LIN {X 0,Y 411.233,Z 499.748,A -85,B 0,C 180,E1 -10713.92,E2 -10713.92} C_VEL
LIN {X 0,Y 411.528,Z 496.938,A -85,B 0,C 180,E1 -10715.39,E2 -10715.39} C_VEL
LIN {X 0,Y 411.956,Z 493.12,A -85,B 0,C 180,E1 -10716.859,E2 -10716.859} C_VEL
LIN {X 0,Y 412.248,Z 487.246,A -85,B 0,C 180,E1 -10718.588,E2 -10718.588} C_VEL
LIN {X 0,Y 412.886,Z 480.826,A -85,B 0,C 180,E1 -10720.048,E2 -10720.048} C_VEL
LIN {X 0,Y 413.463,Z 474.571,A -85,B 0,C 180,E1 -10721.218,E2 -10721.218} C_VEL
LIN {X 0,Y 413.16,Z 470.905,A -85,B 0,C 180,E1 -10721.852,E2 -10721.852} C_VEL
LIN {X 0,Y 410.83,Z 464.808,A -85,B 0,C 180,E1 -10722.887,E2 -10722.887} C_VEL
LIN {X 0,Y 408.489,Z 458.169,A -85,B 0,C 180,E1 -10723.864,E2 -10723.864} C_VEL
LIN {X 0,Y 408.169,Z 453.615,A -85,B 0,C 180,E1 -10724.401,E2 -10724.401} C_VEL
LIN {X 0,Y 408.88,Z 442.463,A -85,B 0,C 180,E1 -10725.449,E2 -10725.449} C_VEL
LIN {X 0,Y 409.109,Z 437.491,A -85,B 0,C 180,E1 -10725.842,E2 -10725.842} C_VEL
LIN {X 0,Y 406.256,Z 427.518,A -85,B 0,C 180,E1 -10726.674,E2 -10726.674} C_VEL
LIN {X 0,Y 404.21,Z 421.137,A -85,B 0,C 180,E1 -10727.15,E2 -10727.15} C_VEL
LIN {X 0,Y 404.167,Z 421.143,A -85,B 0,C 180,E1 -10730.351,E2 -10730.351} C_VEL
LIN {X 0,Y 404.172,Z 421.141,A -85,B 0,C 180,E1 -10733.574,E2 -10733.574} C_VEL
LIN {X 0,Y 404.187,Z 421.137,A -85,B 0,C 180,E1 -10735.766,E2 -10735.766} C_VEL
LIN {X 0,Y 404.198,Z 421.134,A -85,B 0,C 180,E1 -10737.999,E2 -10737.999} C_VEL
LIN {X 0,Y 404.142,Z 421.144,A -85,B 0,C 180,E1 -10741.558,E2 -10741.558} C_VEL
LIN {X 0,Y 404.188,Z 421.14,A -85,B 0,C 180,E1 -10745.016,E2 -10745.016} C_VEL
LIN {X 0,Y 404.167,Z 421.141,A -85,B 0,C 180,E1 -10748.756,E2 -10748.756} C_VEL
LIN {X 0,Y 404.194,Z 421.136,A -85,B 0,C 180,E1 -10751.611,E2 -10751.611} C_VEL
LIN {X 0,Y 404.194,Z 421.136,A -85,B 0,C 180,E1 -10754.529,E2 -10754.529} C_VEL
LIN {X 0,Y 404.142,Z 421.144,A -85,B 0,C 180,E1 -10757.296,E2 -10757.296} C_VEL
LIN {X 0,Y 404.171,Z 421.138,A -85,B 0,C 180,E1 -10759.955,E2 -10759.955} C_VEL
LIN {X 0,Y 404.139,Z 421.146,A -85,B 0,C 180,E1 -10763.125,E2 -10763.125} C_VEL
LIN {X 0,Y 404.147,Z 421.141,A -85,B 0,C 180,E1 -10766.188,E2 -10766.188} C_VEL
LIN {X 0,Y 404.148,Z 421.14,A -85,B 0,C 180,E1 -10769.715,E2 -10769.715} C_VEL
LIN {X 0,Y 404.197,Z 421.137,A -85,B 0,C 180,E1 -10773.123,E2 -10773.123} C_VEL
LIN {X 0,Y 404.179,Z 421.138,A -85,B 0,C 180,E1 -10775.334,E2 -10775.334} C_VEL
LIN {X 0,Y 404.141,Z 421.146,A -85,B 0,C 180,E1 -10778.581,E2 -10778.581} C_VEL
LIN {X 0,Y 404.213,Z 421.132,A -85,B 0,C 180,E1 -10781.762,E2 -10781.762} C_VEL
LIN {X 0,Y 404.211,Z 421.136,A -85,B 0,C 180,E1 -10784.882,E2 -10784.882} C_VEL
LIN {X 0,Y 404.273,Z 421.126,A -85,B 0,C 180,E1 -10787.959,E2 -10787.959} C_VEL
LIN {X 0,Y 404.27,Z 421.127,A -85,B 0,C 180,E1 -10790.998,E2 -10790.998} C_VEL
LIN {X 0,Y 404.421,Z 421.109,A -85,B 0,C 180,E1 -10794.015,E2 -10794.015} C_VEL
LIN {X 0,Y 404.486,Z 421.101,A -85,B 0,C 180,E1 -10798.008,E2 -10798.008} C_VEL
LIN {X 0,Y 404.615,Z 421.084,A -85,B 0,C 180,E1 -10800,E2 -10800} C_VEL
LIN {X 0,Y 404.427,Z 421.107,A -85,B 0,C 180,E1 -10802.988,E2 -10802.988} C_VEL
LIN {X 0,Y 404.421,Z 421.11,A -85,B 0,C 180,E1 -10805.985,E2 -10805.985} C_VEL
LIN {X 0,Y 404.269,Z 421.126,A -85,B 0,C 180,E1 -10809.001,E2 -10809.001} C_VEL
LIN {X 0,Y 404.272,Z 421.129,A -85,B 0,C 180,E1 -10812.041,E2 -10812.041} C_VEL
LIN {X 0,Y 404.211,Z 421.132,A -85,B 0,C 180,E1 -10815.118,E2 -10815.118} C_VEL
LIN {X 0,Y 404.213,Z 421.137,A -85,B 0,C 180,E1 -10818.238,E2 -10818.238} C_VEL
LIN {X 0,Y 404.141,Z 421.142,A -85,B 0,C 180,E1 -10821.419,E2 -10821.419} C_VEL
LIN {X 0,Y 404.176,Z 421.138,A -85,B 0,C 180,E1 -10824.666,E2 -10824.666} C_VEL
LIN {X 0,Y 404.197,Z 421.139,A -85,B 0,C 180,E1 -10828,E2 -10828} C_VEL
LIN {X 0,Y 404.141,Z 421.143,A -85,B 0,C 180,E1 -10831.558,E2 -10831.558} C_VEL
LIN {X 0,Y 404.188,Z 421.136,A -85,B 0,C 180,E1 -10835.016,E2 -10835.016} C_VEL
LIN {X 0,Y 404.16,Z 421.139,A -85,B 0,C 180,E1 -10838.756,E2 -10838.756} C_VEL
LIN {X 0,Y 404.126,Z 421.147,A -85,B 0,C 180,E1 -10841.6,E2 -10841.6} C_VEL
LIN {X 0,Y 404.151,Z 421.147,A -85,B 0,C 180,E1 -10844.523,E2 -10844.523} C_VEL
LIN {X 0,Y 404.173,Z 421.263,A -85,B 0,C 180,E1 -10846.913,E2 -10846.913} C_VEL
LIN {X 0,Y 406.132,Z 430.706,A -85,B 0,C 180,E1 -10850.188,E2 -10850.188} C_VEL
LIN {X 0,Y 407.528,Z 438.986,A -85,B 0,C 180,E1 -10852.872,E2 -10852.872} C_VEL
LIN {X 0,Y 406.783,Z 448.613,A -85,B 0,C 180,E1 -10855.7,E2 -10855.7} C_VEL
LIN {X 0,Y 406.024,Z 460.209,A -85,B 0,C 180,E1 -10859.006,E2 -10859.006} C_VEL
LIN {X 0,Y 405.193,Z 473.421,A -85,B 0,C 180,E1 -10862.679,E2 -10862.679} C_VEL
LIN {X 0,Y 404.587,Z 485.183,A -85,B 0,C 180,E1 -10865.907,E2 -10865.907} C_VEL
LIN {X 0,Y 403.999,Z 498.789,A -85,B 0,C 180,E1 -10869.64,E2 -10869.64} C_VEL
LIN {X 0,Y 403.693,Z 507.433,A -85,B 0,C 180,E1 -10872.033,E2 -10872.033} C_VEL
LIN {X 0,Y 405.431,Z 523.045,A -85,B 0,C 180,E1 -10872.575,E2 -10872.575} C_VEL
LIN {X 0,Y 406.319,Z 535.463,A -85,B 0,C 180,E1 -10873.183,E2 -10873.183} C_VEL
LIN {X 0,Y 406.946,Z 547.554,A -85,B 0,C 180,E1 -10873.959,E2 -10873.959} C_VEL
LIN {X 0,Y 405.977,Z 560.123,A -85,B 0,C 180,E1 -10874.95,E2 -10874.95} C_VEL
LIN {X 0,Y 405.284,Z 570.106,A -85,B 0,C 180,E1 -10875.95,E2 -10875.95} C_VEL
LIN {X 0,Y 404.681,Z 580.266,A -85,B 0,C 180,E1 -10877.207,E2 -10877.207} C_VEL
LIN {X 0,Y 404.04,Z 588.6,A -85,B 0,C 180,E1 -10878.461,E2 -10878.461} C_VEL
LIN {X 0,Y 403.569,Z 596.818,A -85,B 0,C 180,E1 -10879.971,E2 -10879.971} C_VEL
LIN {X 0,Y 403.404,Z 603.456,A -85,B 0,C 180,E1 -10881.484,E2 -10881.484} C_VEL
LIN {X 0,Y 403.35,Z 609.652,A -85,B 0,C 180,E1 -10883.302,E2 -10883.302} C_VEL
LIN {X 0,Y 403.507,Z 613.992,A -85,B 0,C 180,E1 -10885.004,E2 -10885.004} C_VEL
LIN {X 0,Y 403.598,Z 615.936,A -85,B 0,C 180,E1 -10886.006,E2 -10886.006} C_VEL
LIN {X 0,Y 403.567,Z 617.381,A -85,B 0,C 180,E1 -10887.005,E2 -10887.005} C_VEL
LIN {X 0,Y 403.594,Z 618.419,A -85,B 0,C 180,E1 -10888.004,E2 -10888.004} C_VEL
LIN {X 0,Y 403.837,Z 619.307,A -85,B 0,C 180,E1 -10890,E2 -10890} C_VEL
LIN {X 0,Y 403.595,Z 618.417,A -85,B 0,C 180,E1 -10891.996,E2 -10891.996} C_VEL
LIN {X 0,Y 403.567,Z 617.38,A -85,B 0,C 180,E1 -10892.995,E2 -10892.995} C_VEL
LIN {X 0,Y 403.598,Z 615.933,A -85,B 0,C 180,E1 -10893.994,E2 -10893.994} C_VEL
LIN {X 0,Y 403.413,Z 612.861,A -85,B 0,C 180,E1 -10895.498,E2 -10895.498} C_VEL
LIN {X 0,Y 403.354,Z 608.731,A -85,B 0,C 180,E1 -10897.006,E2 -10897.006} C_VEL
LIN {X 0,Y 403.4,Z 602.403,A -85,B 0,C 180,E1 -10898.769,E2 -10898.769} C_VEL
LIN {X 0,Y 403.644,Z 595.53,A -85,B 0,C 180,E1 -10900.281,E2 -10900.281} C_VEL
LIN {X 0,Y 404.114,Z 587.045,A -85,B 0,C 180,E1 -10901.791,E2 -10901.791} C_VEL
LIN {X 0,Y 404.806,Z 578.392,A -85,B 0,C 180,E1 -10903.044,E2 -10903.044} C_VEL
LIN {X 0,Y 405.285,Z 570.06,A -85,B 0,C 180,E1 -10904.05,E2 -10904.05} C_VEL
LIN {X 0,Y 406.099,Z 558.626,A -85,B 0,C 180,E1 -10905.174,E2 -10905.174} C_VEL
LIN {X 0,Y 406.943,Z 547.474,A -85,B 0,C 180,E1 -10906.041,E2 -10906.041} C_VEL
LIN {X 0,Y 406.301,Z 535.359,A -85,B 0,C 180,E1 -10906.818,E2 -10906.818} C_VEL
LIN {X 0,Y 405.431,Z 522.863,A -85,B 0,C 180,E1 -10907.425,E2 -10907.425} C_VEL
LIN {X 0,Y 403.899,Z 509.452,A -85,B 0,C 180,E1 -10907.888,E2 -10907.888} C_VEL
LIN {X 0,Y 403.708,Z 507.4,A -85,B 0,C 180,E1 -10907.966,E2 -10907.966} C_VEL
LIN {X 0,Y 404.129,Z 494.908,A -85,B 0,C 180,E1 -10911.42,E2 -10911.42} C_VEL
LIN {X 0,Y 404.773,Z 481.632,A -85,B 0,C 180,E1 -10915.057,E2 -10915.057} C_VEL
LIN {X 0,Y 405.548,Z 467.226,A -85,B 0,C 180,E1 -10919.028,E2 -10919.028} C_VEL
LIN {X 0,Y 406.352,Z 455.112,A -85,B 0,C 180,E1 -10922.423,E2 -10922.423} C_VEL
LIN {X 0,Y 407.479,Z 440.973,A -85,B 0,C 180,E1 -10926.516,E2 -10926.516} C_VEL
LIN {X 0,Y 407.374,Z 437.82,A -85,B 0,C 180,E1 -10927.478,E2 -10927.478} C_VEL
LIN {X 0,Y 405.818,Z 429.026,A -85,B 0,C 180,E1 -10930.359,E2 -10930.359} C_VEL
LIN {X 0,Y 404.16,Z 421.141,A -85,B 0,C 180,E1 -10933.135,E2 -10933.135} C_VEL
LIN {X 0,Y 404.159,Z 421.144,A -85,B 0,C 180,E1 -10936.916,E2 -10936.916} C_VEL
LIN {X 0,Y 404.171,Z 421.142,A -85,B 0,C 180,E1 -10939.955,E2 -10939.955} C_VEL
LIN {X 0,Y 404.143,Z 421.141,A -85,B 0,C 180,E1 -10943.124,E2 -10943.124} C_VEL
LIN {X 0,Y 404.148,Z 421.145,A -85,B 0,C 180,E1 -10946.188,E2 -10946.188} C_VEL
LIN {X 0,Y 404.149,Z 421.144,A -85,B 0,C 180,E1 -10949.715,E2 -10949.715} C_VEL
LIN {X 0,Y 404.198,Z 421.134,A -85,B 0,C 180,E1 -10953.123,E2 -10953.123} C_VEL
LIN {X 0,Y 404.177,Z 421.138,A -85,B 0,C 180,E1 -10955.334,E2 -10955.334} C_VEL
LIN {X 0,Y 404.142,Z 421.142,A -85,B 0,C 180,E1 -10958.581,E2 -10958.581} C_VEL
LIN {X 0,Y 404.214,Z 421.137,A -85,B 0,C 180,E1 -10961.762,E2 -10961.762} C_VEL
LIN {X 0,Y 404.212,Z 421.132,A -85,B 0,C 180,E1 -10964.882,E2 -10964.882} C_VEL
LIN {X 0,Y 404.273,Z 421.13,A -85,B 0,C 180,E1 -10967.959,E2 -10967.959} C_VEL
LIN {X 0,Y 404.27,Z 421.126,A -85,B 0,C 180,E1 -10970.999,E2 -10970.999} C_VEL
LIN {X 0,Y 404.422,Z 421.11,A -85,B 0,C 180,E1 -10974.015,E2 -10974.015} C_VEL
LIN {X 0,Y 404.487,Z 421.101,A -85,B 0,C 180,E1 -10978.009,E2 -10978.009} C_VEL
LIN {X 0,Y 404.616,Z 421.085,A -85,B 0,C 180,E1 -10980,E2 -10980} C_VEL
LIN {X 0,Y 404.42,Z 421.107,A -85,B 0,C 180,E1 -10982.988,E2 -10982.988} C_VEL
LIN {X 0,Y 404.389,Z 421.111,A -85,B 0,C 180,E1 -10986.642,E2 -10986.642} C_VEL
LIN {X 0,Y 404.265,Z 421.128,A -85,B 0,C 180,E1 -10990.012,E2 -10990.012} C_VEL
LIN {X 0,Y 404.27,Z 421.129,A -85,B 0,C 180,E1 -10993.211,E2 -10993.211} C_VEL
LIN {X 0,Y 404.219,Z 421.134,A -85,B 0,C 180,E1 -10997.007,E2 -10997.007} C_VEL
LIN {X 0,Y 404.167,Z 421.138,A -85,B 0,C 180,E1 -11000.352,E2 -11000.352} C_VEL
LIN {X 0,Y 404.173,Z 421.141,A -85,B 0,C 180,E1 -11003.574,E2 -11003.574} C_VEL
LIN {X 0,Y 404.187,Z 421.138,A -85,B 0,C 180,E1 -11005.766,E2 -11005.766} C_VEL
LIN {X 0,Y 404.199,Z 421.134,A -85,B 0,C 180,E1 -11008,E2 -11008} C_VEL
LIN {X 0,Y 404.143,Z 421.144,A -85,B 0,C 180,E1 -11011.558,E2 -11011.558} C_VEL
LIN {X 0,Y 404.188,Z 421.14,A -85,B 0,C 180,E1 -11015.016,E2 -11015.016} C_VEL
LIN {X 0,Y 404.155,Z 421.142,A -85,B 0,C 180,E1 -11018.757,E2 -11018.757} C_VEL
LIN {X 0,Y 404.127,Z 421.145,A -85,B 0,C 180,E1 -11021.6,E2 -11021.6} C_VEL
LIN {X 0,Y 404.16,Z 421.14,A -85,B 0,C 180,E1 -11024.524,E2 -11024.524} C_VEL
LIN {X 0,Y 404.21,Z 421.137,A -85,B 0,C 180,E1 -11027.305,E2 -11027.305} C_VEL
LIN {X 0,Y 404.172,Z 421.137,A -85,B 0,C 180,E1 -11029.955,E2 -11029.955} C_VEL
LIN {X 0,Y 404.144,Z 421.145,A -85,B 0,C 180,E1 -11033.124,E2 -11033.124} C_VEL
LIN {X 0,Y 404.148,Z 421.141,A -85,B 0,C 180,E1 -11036.188,E2 -11036.188} C_VEL
LIN {X 0,Y 404.149,Z 421.14,A -85,B 0,C 180,E1 -11039.715,E2 -11039.715} C_VEL
LIN {X 0,Y 404.199,Z 421.138,A -85,B 0,C 180,E1 -11043.123,E2 -11043.123} C_VEL
LIN {X 0,Y 404.18,Z 421.138,A -85,B 0,C 180,E1 -11045.334,E2 -11045.334} C_VEL
LIN {X 0,Y 404.142,Z 421.146,A -85,B 0,C 180,E1 -11048.581,E2 -11048.581} C_VEL
LIN {X 0,Y 404.213,Z 421.137,A -85,B 0,C 180,E1 -11051.762,E2 -11051.762} C_VEL
LIN {X 0,Y 404.206,Z 421.138,A -85,B 0,C 180,E1 -11052.951,E2 -11052.951} C_VEL
LIN {X 0,Y 407.905,Z 433.077,A -85,B 0,C 180,E1 -11053.869,E2 -11053.869} C_VEL
LIN {X 0,Y 409.181,Z 438.491,A -85,B 0,C 180,E1 -11054.336,E2 -11054.336} C_VEL
LIN {X 0,Y 408.452,Z 449.646,A -85,B 0,C 180,E1 -11055.298,E2 -11055.298} C_VEL
LIN {X 0,Y 407.754,Z 459.975,A -85,B 0,C 180,E1 -11056.418,E2 -11056.418} C_VEL
LIN {X 0,Y 407.142,Z 468.398,A -85,B 0,C 180,E1 -11057.539,E2 -11057.539} C_VEL
LIN {X 0,Y 406.475,Z 476.152,A -85,B 0,C 180,E1 -11058.784,E2 -11058.784} C_VEL
LIN {X 0,Y 405.752,Z 483.728,A -85,B 0,C 180,E1 -11060.277,E2 -11060.277} C_VEL
LIN {X 0,Y 405.349,Z 488.999,A -85,B 0,C 180,E1 -11061.56,E2 -11061.56} C_VEL
LIN {X 0,Y 405.008,Z 493.848,A -85,B 0,C 180,E1 -11063.023,E2 -11063.023} C_VEL
LIN {X 0,Y 404.54,Z 497.738,A -85,B 0,C 180,E1 -11064.517,E2 -11064.517} C_VEL
LIN {X 0,Y 404.23,Z 500.603,A -85,B 0,C 180,E1 -11066.012,E2 -11066.012} C_VEL
LIN {X 0,Y 404.065,Z 501.98,A -85,B 0,C 180,E1 -11067.009,E2 -11067.009} C_VEL
LIN {X 0,Y 404.047,Z 503.535,A -85,B 0,C 180,E1 -11069.003,E2 -11069.003} C_VEL
LIN {X 0,Y 404.094,Z 503.755,A -85,B 0,C 180,E1 -11070,E2 -11070} C_VEL
LIN {X 0,Y 404.077,Z 503.012,A -85,B 0,C 180,E1 -11071.993,E2 -11071.993} C_VEL
LIN {X 0,Y 404.059,Z 502.083,A -85,B 0,C 180,E1 -11072.991,E2 -11072.991} C_VEL
LIN {X 0,Y 404.221,Z 500.753,A -85,B 0,C 180,E1 -11073.988,E2 -11073.988} C_VEL
LIN {X 0,Y 404.534,Z 497.942,A -85,B 0,C 180,E1 -11075.483,E2 -11075.483} C_VEL
LIN {X 0,Y 404.98,Z 494.123,A -85,B 0,C 180,E1 -11076.977,E2 -11076.977} C_VEL
LIN {X 0,Y 405.3,Z 488.249,A -85,B 0,C 180,E1 -11078.736,E2 -11078.736} C_VEL
LIN {X 0,Y 405.969,Z 481.829,A -85,B 0,C 180,E1 -11080.221,E2 -11080.221} C_VEL
LIN {X 0,Y 406.706,Z 473.805,A -85,B 0,C 180,E1 -11081.715,E2 -11081.715} C_VEL
LIN {X 0,Y 407.321,Z 465.586,A -85,B 0,C 180,E1 -11082.962,E2 -11082.962} C_VEL
LIN {X 0,Y 408.066,Z 455.402,A -85,B 0,C 180,E1 -11084.207,E2 -11084.207} C_VEL
LIN {X 0,Y 408.169,Z 453.615,A -85,B 0,C 180,E1 -11084.401,E2 -11084.401} C_VEL
LIN {X 0,Y 407.815,Z 448.942,A -85,B 0,C 180,E1 -11084.911,E2 -11084.911} C_VEL
LIN {X 0,Y 406.388,Z 444.383,A -85,B 0,C 180,E1 -11085.415,E2 -11085.415} C_VEL
LIN {X 0,Y 402.042,Z 435.304,A -85,B 0,C 180,E1 -11086.372,E2 -11086.372} C_VEL
LIN {X 0,Y 399.35,Z 428.824,A -85,B 0,C 180,E1 -11086.954,E2 -11086.954} C_VEL
LIN {X 0,Y 397.163,Z 422.015,A -85,B 0,C 180,E1 -11087.475,E2 -11087.475} C_VEL
LIN {X 0,Y 397.105,Z 422.021,A -85,B 0,C 180,E1 -11090.73,E2 -11090.73} C_VEL
LIN {X 0,Y 397.136,Z 422.014,A -85,B 0,C 180,E1 -11094.018,E2 -11094.018} C_VEL
LIN {X 0,Y 397.197,Z 422.011,A -85,B 0,C 180,E1 -11097.39,E2 -11097.39} C_VEL
LIN {X 0,Y 397.081,Z 422.024,A -85,B 0,C 180,E1 -11100.882,E2 -11100.882} C_VEL
LIN {X 0,Y 397.129,Z 422.015,A -85,B 0,C 180,E1 -11104.493,E2 -11104.493} C_VEL
LIN {X 0,Y 397.113,Z 422.017,A -85,B 0,C 180,E1 -11108.274,E2 -11108.274} C_VEL
LIN {X 0,Y 397.159,Z 422.011,A -85,B 0,C 180,E1 -11111.993,E2 -11111.993} C_VEL
LIN {X 0,Y 397.117,Z 422.021,A -85,B 0,C 180,E1 -11115.065,E2 -11115.065} C_VEL
LIN {X 0,Y 397.07,Z 422.022,A -85,B 0,C 180,E1 -11118.021,E2 -11118.021} C_VEL
LIN {X 0,Y 397.133,Z 422.019,A -85,B 0,C 180,E1 -11121.138,E2 -11121.138} C_VEL
LIN {X 0,Y 397.121,Z 422.018,A -85,B 0,C 180,E1 -11124.497,E2 -11124.497} C_VEL
LIN {X 0,Y 397.08,Z 422.02,A -85,B 0,C 180,E1 -11127.928,E2 -11127.928} C_VEL
LIN {X 0,Y 397.124,Z 422.016,A -85,B 0,C 180,E1 -11131.456,E2 -11131.456} C_VEL
LIN {X 0,Y 397.155,Z 422.015,A -85,B 0,C 180,E1 -11134.488,E2 -11134.488} C_VEL
LIN {X 0,Y 397.111,Z 422.02,A -85,B 0,C 180,E1 -11137.086,E2 -11137.086} C_VEL
LIN {X 0,Y 397.151,Z 422.015,A -85,B 0,C 180,E1 -11140.353,E2 -11140.353} C_VEL
LIN {X 0,Y 397.169,Z 422.009,A -85,B 0,C 180,E1 -11143.553,E2 -11143.553} C_VEL
LIN {X 0,Y 397.231,Z 422.007,A -85,B 0,C 180,E1 -11146.703,E2 -11146.703} C_VEL
LIN {X 0,Y 397.224,Z 422.003,A -85,B 0,C 180,E1 -11149.809,E2 -11149.809} C_VEL
LIN {X 0,Y 397.341,Z 421.991,A -85,B 0,C 180,E1 -11152.888,E2 -11152.888} C_VEL
LIN {X 0,Y 397.256,Z 422.001,A -85,B 0,C 180,E1 -11154.925,E2 -11154.925} C_VEL
LIN {X 0,Y 397.455,Z 421.976,A -85,B 0,C 180,E1 -11157.973,E2 -11157.973} C_VEL
LIN {X 0,Y 397.584,Z 421.96,A -85,B 0,C 180,E1 -11160,E2 -11160} C_VEL
LIN {X 0,Y 397.385,Z 421.983,A -85,B 0,C 180,E1 -11163.041,E2 -11163.041} C_VEL
LIN {X 0,Y 397.371,Z 421.989,A -85,B 0,C 180,E1 -11166.092,E2 -11166.092} C_VEL
LIN {X 0,Y 397.239,Z 422.001,A -85,B 0,C 180,E1 -11169.162,E2 -11169.162} C_VEL
LIN {X 0,Y 397.231,Z 422.007,A -85,B 0,C 180,E1 -11172.258,E2 -11172.258} C_VEL
LIN {X 0,Y 397.183,Z 422.008,A -85,B 0,C 180,E1 -11175.392,E2 -11175.392} C_VEL
LIN {X 0,Y 397.165,Z 422.013,A -85,B 0,C 180,E1 -11178.573,E2 -11178.573} C_VEL
LIN {X 0,Y 397.098,Z 422.022,A -85,B 0,C 180,E1 -11181.818,E2 -11181.818} C_VEL
LIN {X 0,Y 397.154,Z 422.013,A -85,B 0,C 180,E1 -11185.512,E2 -11185.512} C_VEL
LIN {X 0,Y 397.124,Z 422.017,A -85,B 0,C 180,E1 -11188.544,E2 -11188.544} C_VEL
LIN {X 0,Y 397.081,Z 422.026,A -85,B 0,C 180,E1 -11192.071,E2 -11192.071} C_VEL
LIN {X 0,Y 397.122,Z 422.018,A -85,B 0,C 180,E1 -11195.504,E2 -11195.504} C_VEL
LIN {X 0,Y 397.135,Z 422.014,A -85,B 0,C 180,E1 -11198.862,E2 -11198.862} C_VEL
LIN {X 0,Y 397.073,Z 422.029,A -85,B 0,C 180,E1 -11202.267,E2 -11202.267} C_VEL
LIN {X 0,Y 397.091,Z 422.026,A -85,B 0,C 180,E1 -11205.068,E2 -11205.068} C_VEL
LIN {X 0,Y 397.104,Z 422.073,A -85,B 0,C 180,E1 -11206.521,E2 -11206.521} C_VEL
LIN {X 0,Y 399.138,Z 431.9,A -85,B 0,C 180,E1 -11210.007,E2 -11210.007} C_VEL
LIN {X 0,Y 400.585,Z 440.329,A -85,B 0,C 180,E1 -11212.798,E2 -11212.798} C_VEL
LIN {X 0,Y 399.688,Z 451.265,A -85,B 0,C 180,E1 -11216.063,E2 -11216.063} C_VEL
LIN {X 0,Y 398.92,Z 462.345,A -85,B 0,C 180,E1 -11219.276,E2 -11219.276} C_VEL
LIN {X 0,Y 398.123,Z 474.34,A -85,B 0,C 180,E1 -11222.679,E2 -11222.679} C_VEL
LIN {X 0,Y 397.501,Z 486.179,A -85,B 0,C 180,E1 -11226.005,E2 -11226.005} C_VEL
LIN {X 0,Y 396.882,Z 499.716,A -85,B 0,C 180,E1 -11229.806,E2 -11229.806} C_VEL
LIN {X 0,Y 396.646,Z 506.407,A -85,B 0,C 180,E1 -11231.703,E2 -11231.703} C_VEL
LIN {X 0,Y 398.444,Z 522.202,A -85,B 0,C 180,E1 -11232.267,E2 -11232.267} C_VEL
LIN {X 0,Y 399.331,Z 535.112,A -85,B 0,C 180,E1 -11232.919,E2 -11232.919} C_VEL
LIN {X 0,Y 399.963,Z 548.32,A -85,B 0,C 180,E1 -11233.803,E2 -11233.803} C_VEL
LIN {X 0,Y 399.091,Z 559.106,A -85,B 0,C 180,E1 -11234.684,E2 -11234.684} C_VEL
LIN {X 0,Y 398.342,Z 569.085,A -85,B 0,C 180,E1 -11235.7,E2 -11235.7} C_VEL
LIN {X 0,Y 397.739,Z 577.395,A -85,B 0,C 180,E1 -11236.72,E2 -11236.72} C_VEL
LIN {X 0,Y 397.08,Z 586.048,A -85,B 0,C 180,E1 -11237.997,E2 -11237.997} C_VEL
LIN {X 0,Y 396.584,Z 594.528,A -85,B 0,C 180,E1 -11239.535,E2 -11239.535} C_VEL
LIN {X 0,Y 396.35,Z 601.402,A -85,B 0,C 180,E1 -11241.074,E2 -11241.074} C_VEL
LIN {X 0,Y 396.289,Z 607.727,A -85,B 0,C 180,E1 -11242.869,E2 -11242.869} C_VEL
LIN {X 0,Y 396.343,Z 611.853,A -85,B 0,C 180,E1 -11244.403,E2 -11244.403} C_VEL
LIN {X 0,Y 396.559,Z 614.927,A -85,B 0,C 180,E1 -11245.935,E2 -11245.935} C_VEL
LIN {X 0,Y 396.525,Z 616.373,A -85,B 0,C 180,E1 -11246.952,E2 -11246.952} C_VEL
LIN {X 0,Y 396.555,Z 617.411,A -85,B 0,C 180,E1 -11247.969,E2 -11247.969} C_VEL
LIN {X 0,Y 396.813,Z 618.303,A -85,B 0,C 180,E1 -11250,E2 -11250} C_VEL
LIN {X 0,Y 396.556,Z 617.41,A -85,B 0,C 180,E1 -11252.031,E2 -11252.031} C_VEL
LIN {X 0,Y 396.525,Z 616.371,A -85,B 0,C 180,E1 -11253.048,E2 -11253.048} C_VEL
LIN {X 0,Y 396.559,Z 614.923,A -85,B 0,C 180,E1 -11254.065,E2 -11254.065} C_VEL
LIN {X 0,Y 396.341,Z 611.844,A -85,B 0,C 180,E1 -11255.597,E2 -11255.597} C_VEL
LIN {X 0,Y 396.291,Z 607.712,A -85,B 0,C 180,E1 -11257.131,E2 -11257.131} C_VEL
LIN {X 0,Y 396.35,Z 601.381,A -85,B 0,C 180,E1 -11258.926,E2 -11258.926} C_VEL
LIN {X 0,Y 396.59,Z 594.503,A -85,B 0,C 180,E1 -11260.466,E2 -11260.466} C_VEL
LIN {X 0,Y 397.073,Z 586.014,A -85,B 0,C 180,E1 -11262.004,E2 -11262.004} C_VEL
LIN {X 0,Y 397.742,Z 577.352,A -85,B 0,C 180,E1 -11263.28,E2 -11263.28} C_VEL
LIN {X 0,Y 398.461,Z 567.875,A -85,B 0,C 180,E1 -11264.426,E2 -11264.426} C_VEL
LIN {X 0,Y 399.219,Z 557.602,A -85,B 0,C 180,E1 -11265.442,E2 -11265.442} C_VEL
LIN {X 0,Y 399.97,Z 548.234,A -85,B 0,C 180,E1 -11266.197,E2 -11266.197} C_VEL
LIN {X 0,Y 399.378,Z 536.08,A -85,B 0,C 180,E1 -11267.017,E2 -11267.017} C_VEL
LIN {X 0,Y 398.484,Z 522.427,A -85,B 0,C 180,E1 -11267.715,E2 -11267.715} C_VEL
LIN {X 0,Y 396.969,Z 509.154,A -85,B 0,C 180,E1 -11268.194,E2 -11268.194} C_VEL
LIN {X 0,Y 396.663,Z 506.375,A -85,B 0,C 180,E1 -11268.297,E2 -11268.297} C_VEL
LIN {X 0,Y 397.105,Z 493.918,A -85,B 0,C 180,E1 -11271.818,E2 -11271.818} C_VEL
LIN {X 0,Y 397.768,Z 481.132,A -85,B 0,C 180,E1 -11275.401,E2 -11275.401} C_VEL
LIN {X 0,Y 398.542,Z 467.315,A -85,B 0,C 180,E1 -11279.298,E2 -11279.298} C_VEL
LIN {X 0,Y 399.391,Z 455.629,A -85,B 0,C 180,E1 -11282.647,E2 -11282.647} C_VEL
LIN {X 0,Y 400.523,Z 442.162,A -85,B 0,C 180,E1 -11286.627,E2 -11286.627} C_VEL
LIN {X 0,Y 400.268,Z 438.058,A -85,B 0,C 180,E1 -11287.919,E2 -11287.919} C_VEL
LIN {X 0,Y 398.708,Z 429.741,A -85,B 0,C 180,E1 -11290.715,E2 -11290.715} C_VEL
LIN {X 0,Y 397.113,Z 422.017,A -85,B 0,C 180,E1 -11293.52,E2 -11293.52} C_VEL
LIN {X 0,Y 397.107,Z 422.023,A -85,B 0,C 180,E1 -11296.521,E2 -11296.521} C_VEL
LIN {X 0,Y 397.117,Z 422.02,A -85,B 0,C 180,E1 -11300.423,E2 -11300.423} C_VEL
LIN {X 0,Y 397.112,Z 422.021,A -85,B 0,C 180,E1 -11304.266,E2 -11304.266} C_VEL
LIN {X 0,Y 397.117,Z 422.017,A -85,B 0,C 180,E1 -11306.727,E2 -11306.727} C_VEL
LIN {X 0,Y 397.127,Z 422.018,A -85,B 0,C 180,E1 -11310.296,E2 -11310.296} C_VEL
LIN {X 0,Y 397.197,Z 422.007,A -85,B 0,C 180,E1 -11312.61,E2 -11312.61} C_VEL
LIN {X 0,Y 397.131,Z 422.019,A -85,B 0,C 180,E1 -11315.982,E2 -11315.982} C_VEL
LIN {X 0,Y 397.142,Z 422.017,A -85,B 0,C 180,E1 -11319.705,E2 -11319.705} C_VEL
LIN {X 0,Y 397.185,Z 422.007,A -85,B 0,C 180,E1 -11322.845,E2 -11322.845} C_VEL
LIN {X 0,Y 397.23,Z 422.002,A -85,B 0,C 180,E1 -11326.679,E2 -11326.679} C_VEL
LIN {X 0,Y 397.224,Z 422.008,A -85,B 0,C 180,E1 -11329.809,E2 -11329.809} C_VEL
LIN {X 0,Y 397.341,Z 421.988,A -85,B 0,C 180,E1 -11332.888,E2 -11332.888} C_VEL
LIN {X 0,Y 397.259,Z 421.999,A -85,B 0,C 180,E1 -11334.925,E2 -11334.925} C_VEL
LIN {X 0,Y 397.456,Z 421.977,A -85,B 0,C 180,E1 -11337.973,E2 -11337.973} C_VEL
LIN {X 0,Y 397.585,Z 421.96,A -85,B 0,C 180,E1 -11340,E2 -11340} C_VEL
LIN {X 0,Y 397.38,Z 421.985,A -85,B 0,C 180,E1 -11343.041,E2 -11343.041} C_VEL
LIN {X 0,Y 397.339,Z 421.988,A -85,B 0,C 180,E1 -11346.639,E2 -11346.639} C_VEL
LIN {X 0,Y 397.226,Z 422.003,A -85,B 0,C 180,E1 -11350.191,E2 -11350.191} C_VEL
LIN {X 0,Y 397.23,Z 422.007,A -85,B 0,C 180,E1 -11353.321,E2 -11353.321} C_VEL
LIN {X 0,Y 397.185,Z 422.011,A -85,B 0,C 180,E1 -11357.155,E2 -11357.155} C_VEL
LIN {X 0,Y 397.112,Z 422.018,A -85,B 0,C 180,E1 -11360.73,E2 -11360.73} C_VEL
LIN {X 0,Y 397.136,Z 422.014,A -85,B 0,C 180,E1 -11364.018,E2 -11364.018} C_VEL
LIN {X 0,Y 397.198,Z 422.011,A -85,B 0,C 180,E1 -11367.39,E2 -11367.39} C_VEL
LIN {X 0,Y 397.082,Z 422.023,A -85,B 0,C 180,E1 -11370.882,E2 -11370.882} C_VEL
LIN {X 0,Y 397.128,Z 422.015,A -85,B 0,C 180,E1 -11374.493,E2 -11374.493} C_VEL
LIN {X 0,Y 397.104,Z 422.018,A -85,B 0,C 180,E1 -11378.275,E2 -11378.275} C_VEL
LIN {X 0,Y 397.092,Z 422.024,A -85,B 0,C 180,E1 -11380.909,E2 -11380.909} C_VEL
LIN {X 0,Y 397.108,Z 422.018,A -85,B 0,C 180,E1 -11383.648,E2 -11383.648} C_VEL
LIN {X 0,Y 397.163,Z 422.012,A -85,B 0,C 180,E1 -11386.512,E2 -11386.512} C_VEL
LIN {X 0,Y 397.127,Z 422.016,A -85,B 0,C 180,E1 -11389.551,E2 -11389.551} C_VEL
LIN {X 0,Y 397.102,Z 422.022,A -85,B 0,C 180,E1 -11392.79,E2 -11392.79} C_VEL
LIN {X 0,Y 397.121,Z 422.016,A -85,B 0,C 180,E1 -11396.282,E2 -11396.282} C_VEL
LIN {X 0,Y 397.108,Z 422.017,A -85,B 0,C 180,E1 -11400.135,E2 -11400.135} C_VEL
LIN {X 0,Y 397.198,Z 422.01,A -85,B 0,C 180,E1 -11402.61,E2 -11402.61} C_VEL
LIN {X 0,Y 397.136,Z 422.014,A -85,B 0,C 180,E1 -11405.982,E2 -11405.982} C_VEL
LIN {X 0,Y 397.142,Z 422.013,A -85,B 0,C 180,E1 -11409.705,E2 -11409.705} C_VEL
LIN {X 0,Y 397.192,Z 422.21,A -85,B 0,C 180,E1 -11412.655,E2 -11412.655} C_VEL
LIN {X 0,Y 400.739,Z 433.442,A -85,B 0,C 180,E1 -11413.525,E2 -11413.525} C_VEL
LIN {X 0,Y 402.407,Z 439.717,A -85,B 0,C 180,E1 -11414.083,E2 -11414.083} C_VEL
LIN {X 0,Y 401.666,Z 450.654,A -85,B 0,C 180,E1 -11415.044,E2 -11415.044} C_VEL
LIN {X 0,Y 400.927,Z 460.984,A -85,B 0,C 180,E1 -11416.182,E2 -11416.182} C_VEL
LIN {X 0,Y 400.285,Z 469.406,A -85,B 0,C 180,E1 -11417.322,E2 -11417.322} C_VEL
LIN {X 0,Y 399.588,Z 477.159,A -85,B 0,C 180,E1 -11418.588,E2 -11418.588} C_VEL
LIN {X 0,Y 398.827,Z 484.735,A -85,B 0,C 180,E1 -11420.107,E2 -11420.107} C_VEL
LIN {X 0,Y 398.399,Z 490.005,A -85,B 0,C 180,E1 -11421.412,E2 -11421.412} C_VEL
LIN {X 0,Y 398.035,Z 494.854,A -85,B 0,C 180,E1 -11422.9,E2 -11422.9} C_VEL
LIN {X 0,Y 397.547,Z 498.744,A -85,B 0,C 180,E1 -11424.42,E2 -11424.42} C_VEL
LIN {X 0,Y 397.219,Z 501.609,A -85,B 0,C 180,E1 -11425.942,E2 -11425.942} C_VEL
LIN {X 0,Y 397.047,Z 502.986,A -85,B 0,C 180,E1 -11426.956,E2 -11426.956} C_VEL
LIN {X 0,Y 397.041,Z 504.538,A -85,B 0,C 180,E1 -11428.986,E2 -11428.986} C_VEL
LIN {X 0,Y 397.079,Z 504.759,A -85,B 0,C 180,E1 -11430,E2 -11430} C_VEL
LIN {X 0,Y 397.055,Z 504.016,A -85,B 0,C 180,E1 -11432.029,E2 -11432.029} C_VEL
LIN {X 0,Y 397.041,Z 503.087,A -85,B 0,C 180,E1 -11433.044,E2 -11433.044} C_VEL
LIN {X 0,Y 397.21,Z 501.757,A -85,B 0,C 180,E1 -11434.058,E2 -11434.058} C_VEL
LIN {X 0,Y 397.542,Z 498.946,A -85,B 0,C 180,E1 -11435.58,E2 -11435.58} C_VEL
LIN {X 0,Y 398.006,Z 495.127,A -85,B 0,C 180,E1 -11437.1,E2 -11437.1} C_VEL
LIN {X 0,Y 398.355,Z 489.253,A -85,B 0,C 180,E1 -11438.89,E2 -11438.89} C_VEL
LIN {X 0,Y 399.055,Z 482.832,A -85,B 0,C 180,E1 -11440.4,E2 -11440.4} C_VEL
LIN {X 0,Y 399.835,Z 474.806,A -85,B 0,C 180,E1 -11441.919,E2 -11441.919} C_VEL
LIN {X 0,Y 400.475,Z 466.588,A -85,B 0,C 180,E1 -11443.188,E2 -11443.188} C_VEL
LIN {X 0,Y 401.256,Z 456.403,A -85,B 0,C 180,E1 -11444.453,E2 -11444.453} C_VEL
LIN {X 0,Y 402.052,Z 445.097,A -85,B 0,C 180,E1 -11445.571,E2 -11445.571} C_VEL
LIN {X 0,Y 402.278,Z 439.021,A -85,B 0,C 180,E1 -11446.079,E2 -11446.079} C_VEL
LIN {X 0,Y 399.35,Z 428.824,A -85,B 0,C 180,E1 -11446.954,E2 -11446.954} C_VEL
LIN {X 0,Y 398.113,Z 426.123,A -85,B 0,C 180,E1 -11447.286,E2 -11447.286} C_VEL
LIN {X 0,Y 396.641,Z 424.29,A -85,B 0,C 180,E1 -11447.718,E2 -11447.718} C_VEL
LIN {X 0,Y 394.36,Z 422.824,A -85,B 0,C 180,E1 -11448.473,E2 -11448.473} C_VEL
LIN {X 0,Y 392.277,Z 422.624,A -85,B 0,C 180,E1 -11449.323,E2 -11449.323} C_VEL
LIN {X 0,Y 390.372,Z 422.877,A -85,B 0,C 180,E1 -11450.532,E2 -11450.532} C_VEL
LIN {X 0,Y 390.056,Z 422.899,A -85,B 0,C 180,E1 -11451.152,E2 -11451.152} C_VEL
LIN {X 0,Y 390.083,Z 422.892,A -85,B 0,C 180,E1 -11454.481,E2 -11454.481} C_VEL
LIN {X 0,Y 390.12,Z 422.888,A -85,B 0,C 180,E1 -11457.93,E2 -11457.93} C_VEL
LIN {X 0,Y 390.026,Z 422.902,A -85,B 0,C 180,E1 -11461.504,E2 -11461.504} C_VEL
LIN {X 0,Y 390.071,Z 422.894,A -85,B 0,C 180,E1 -11464.025,E2 -11464.025} C_VEL
LIN {X 0,Y 390.05,Z 422.898,A -85,B 0,C 180,E1 -11467.552,E2 -11467.552} C_VEL
LIN {X 0,Y 390.086,Z 422.896,A -85,B 0,C 180,E1 -11470.826,E2 -11470.826} C_VEL
LIN {X 0,Y 390.107,Z 422.889,A -85,B 0,C 180,E1 -11473.894,E2 -11473.894} C_VEL
LIN {X 0,Y 390.047,Z 422.897,A -85,B 0,C 180,E1 -11477.625,E2 -11477.625} C_VEL
LIN {X 0,Y 390.093,Z 422.897,A -85,B 0,C 180,E1 -11480.908,E2 -11480.908} C_VEL
LIN {X 0,Y 390.087,Z 422.897,A -85,B 0,C 180,E1 -11484.793,E2 -11484.793} C_VEL
LIN {X 0,Y 390.026,Z 422.902,A -85,B 0,C 180,E1 -11488.496,E2 -11488.496} C_VEL
LIN {X 0,Y 390.119,Z 422.888,A -85,B 0,C 180,E1 -11492.07,E2 -11492.07} C_VEL
LIN {X 0,Y 390.081,Z 422.893,A -85,B 0,C 180,E1 -11495.519,E2 -11495.519} C_VEL
LIN {X 0,Y 390.058,Z 422.9,A -85,B 0,C 180,E1 -11498.878,E2 -11498.878} C_VEL
LIN {X 0,Y 390.131,Z 422.888,A -85,B 0,C 180,E1 -11502.167,E2 -11502.167} C_VEL
LIN {X 0,Y 390.15,Z 422.884,A -85,B 0,C 180,E1 -11505.393,E2 -11505.393} C_VEL
LIN {X 0,Y 390.161,Z 422.888,A -85,B 0,C 180,E1 -11508.571,E2 -11508.571} C_VEL
LIN {X 0,Y 390.272,Z 422.871,A -85,B 0,C 180,E1 -11512.071,E2 -11512.071} C_VEL
LIN {X 0,Y 390.228,Z 422.877,A -85,B 0,C 180,E1 -11514.833,E2 -11514.833} C_VEL
LIN {X 0,Y 390.423,Z 422.851,A -85,B 0,C 180,E1 -11517.937,E2 -11517.937} C_VEL
LIN {X 0,Y 390.553,Z 422.836,A -85,B 0,C 180,E1 -11520,E2 -11520} C_VEL
LIN {X 0,Y 390.319,Z 422.863,A -85,B 0,C 180,E1 -11523.096,E2 -11523.096} C_VEL
LIN {X 0,Y 390.324,Z 422.867,A -85,B 0,C 180,E1 -11526.202,E2 -11526.202} C_VEL
LIN {X 0,Y 390.197,Z 422.878,A -85,B 0,C 180,E1 -11529.329,E2 -11529.329} C_VEL
LIN {X 0,Y 390.18,Z 422.884,A -85,B 0,C 180,E1 -11532.483,E2 -11532.483} C_VEL
LIN {X 0,Y 390.142,Z 422.886,A -85,B 0,C 180,E1 -11535.677,E2 -11535.677} C_VEL
LIN {X 0,Y 390.108,Z 422.889,A -85,B 0,C 180,E1 -11538.922,E2 -11538.922} C_VEL
LIN {X 0,Y 390.04,Z 422.902,A -85,B 0,C 180,E1 -11542.234,E2 -11542.234} C_VEL
LIN {X 0,Y 390.121,Z 422.89,A -85,B 0,C 180,E1 -11545.743,E2 -11545.743} C_VEL
LIN {X 0,Y 390.06,Z 422.895,A -85,B 0,C 180,E1 -11549.109,E2 -11549.109} C_VEL
LIN {X 0,Y 390.045,Z 422.897,A -85,B 0,C 180,E1 -11552.721,E2 -11552.721} C_VEL
LIN {X 0,Y 390.059,Z 422.9,A -85,B 0,C 180,E1 -11555.826,E2 -11555.826} C_VEL
LIN {X 0,Y 390.073,Z 422.894,A -85,B 0,C 180,E1 -11559.219,E2 -11559.219} C_VEL
LIN {X 0,Y 390.047,Z 422.905,A -85,B 0,C 180,E1 -11562.375,E2 -11562.375} C_VEL
LIN {X 0,Y 390.047,Z 422.9,A -85,B 0,C 180,E1 -11565.355,E2 -11565.355} C_VEL
LIN {X 0,Y 390.057,Z 423.017,A -85,B 0,C 180,E1 -11566.163,E2 -11566.163} C_VEL
LIN {X 0,Y 391.921,Z 431.761,A -85,B 0,C 180,E1 -11569.362,E2 -11569.362} C_VEL
LIN {X 0,Y 393.459,Z 440.183,A -85,B 0,C 180,E1 -11572.236,E2 -11572.236} C_VEL
LIN {X 0,Y 393.47,Z 444.145,A -85,B 0,C 180,E1 -11573.492,E2 -11573.492} C_VEL
LIN {X 0,Y 392.34,Z 457.436,A -85,B 0,C 180,E1 -11577.494,E2 -11577.494} C_VEL
LIN {X 0,Y 391.432,Z 469.433,A -85,B 0,C 180,E1 -11581.002,E2 -11581.002} C_VEL
LIN {X 0,Y 390.727,Z 481.302,A -85,B 0,C 180,E1 -11584.425,E2 -11584.425} C_VEL
LIN {X 0,Y 390.083,Z 492.957,A -85,B 0,C 180,E1 -11587.768,E2 -11587.768} C_VEL
LIN {X 0,Y 389.594,Z 505.379,A -85,B 0,C 180,E1 -11591.36,E2 -11591.36} C_VEL
LIN {X 0,Y 391.498,Z 521.555,A -85,B 0,C 180,E1 -11591.958,E2 -11591.958} C_VEL
LIN {X 0,Y 392.366,Z 534.759,A -85,B 0,C 180,E1 -11592.646,E2 -11592.646} C_VEL
LIN {X 0,Y 392.933,Z 547.277,A -85,B 0,C 180,E1 -11593.505,E2 -11593.505} C_VEL
LIN {X 0,Y 392.367,Z 556.656,A -85,B 0,C 180,E1 -11594.281,E2 -11594.281} C_VEL
LIN {X 0,Y 391.533,Z 566.911,A -85,B 0,C 180,E1 -11595.313,E2 -11595.313} C_VEL
LIN {X 0,Y 390.722,Z 576.365,A -85,B 0,C 180,E1 -11596.477,E2 -11596.477} C_VEL
LIN {X 0,Y 390.204,Z 583.403,A -85,B 0,C 180,E1 -11597.518,E2 -11597.518} C_VEL
LIN {X 0,Y 389.619,Z 592.238,A -85,B 0,C 180,E1 -11599.082,E2 -11599.082} C_VEL
LIN {X 0,Y 389.336,Z 599.339,A -85,B 0,C 180,E1 -11600.65,E2 -11600.65} C_VEL
LIN {X 0,Y 389.223,Z 605.056,A -85,B 0,C 180,E1 -11602.217,E2 -11602.217} C_VEL
LIN {X 0,Y 389.274,Z 609.566,A -85,B 0,C 180,E1 -11603.781,E2 -11603.781} C_VEL
LIN {X 0,Y 389.351,Z 611.961,A -85,B 0,C 180,E1 -11604.822,E2 -11604.822} C_VEL
LIN {X 0,Y 389.5,Z 613.916,A -85,B 0,C 180,E1 -11605.861,E2 -11605.861} C_VEL
LIN {X 0,Y 389.482,Z 615.364,A -85,B 0,C 180,E1 -11606.897,E2 -11606.897} C_VEL
LIN {X 0,Y 389.515,Z 616.404,A -85,B 0,C 180,E1 -11607.932,E2 -11607.932} C_VEL
LIN {X 0,Y 389.787,Z 617.298,A -85,B 0,C 180,E1 -11610,E2 -11610} C_VEL
LIN {X 0,Y 389.516,Z 616.402,A -85,B 0,C 180,E1 -11612.068,E2 -11612.068} C_VEL
LIN {X 0,Y 389.483,Z 615.362,A -85,B 0,C 180,E1 -11613.103,E2 -11613.103} C_VEL
LIN {X 0,Y 389.5,Z 613.911,A -85,B 0,C 180,E1 -11614.139,E2 -11614.139} C_VEL
LIN {X 0,Y 389.272,Z 610.827,A -85,B 0,C 180,E1 -11615.699,E2 -11615.699} C_VEL
LIN {X 0,Y 389.226,Z 606.692,A -85,B 0,C 180,E1 -11617.261,E2 -11617.261} C_VEL
LIN {X 0,Y 389.301,Z 600.359,A -85,B 0,C 180,E1 -11619.089,E2 -11619.089} C_VEL
LIN {X 0,Y 389.557,Z 593.478,A -85,B 0,C 180,E1 -11620.657,E2 -11620.657} C_VEL
LIN {X 0,Y 390.048,Z 584.984,A -85,B 0,C 180,E1 -11622.223,E2 -11622.223} C_VEL
LIN {X 0,Y 390.672,Z 578.169,A -85,B 0,C 180,E1 -11623.26,E2 -11623.26} C_VEL
LIN {X 0,Y 391.311,Z 569.144,A -85,B 0,C 180,E1 -11624.424,E2 -11624.424} C_VEL
LIN {X 0,Y 392.214,Z 558.017,A -85,B 0,C 180,E1 -11625.592,E2 -11625.592} C_VEL
LIN {X 0,Y 393.004,Z 548.931,A -85,B 0,C 180,E1 -11626.359,E2 -11626.359} C_VEL
LIN {X 0,Y 392.46,Z 536.664,A -85,B 0,C 180,E1 -11627.231,E2 -11627.231} C_VEL
LIN {X 0,Y 391.647,Z 523.328,A -85,B 0,C 180,E1 -11627.95,E2 -11627.95} C_VEL
LIN {X 0,Y 390.189,Z 510.041,A -85,B 0,C 180,E1 -11628.476,E2 -11628.476} C_VEL
LIN {X 0,Y 389.607,Z 505.334,A -85,B 0,C 180,E1 -11628.64,E2 -11628.64} C_VEL
LIN {X 0,Y 390.084,Z 492.925,A -85,B 0,C 180,E1 -11632.232,E2 -11632.232} C_VEL
LIN {X 0,Y 390.728,Z 481.256,A -85,B 0,C 180,E1 -11635.575,E2 -11635.575} C_VEL
LIN {X 0,Y 391.439,Z 469.377,A -85,B 0,C 180,E1 -11638.997,E2 -11638.997} C_VEL
LIN {X 0,Y 392.379,Z 456.853,A -85,B 0,C 180,E1 -11642.666,E2 -11642.666} C_VEL
LIN {X 0,Y 393.473,Z 444.091,A -85,B 0,C 180,E1 -11646.509,E2 -11646.509} C_VEL
LIN {X 0,Y 393.398,Z 440.135,A -85,B 0,C 180,E1 -11647.766,E2 -11647.766} C_VEL
LIN {X 0,Y 391.897,Z 431.729,A -85,B 0,C 180,E1 -11650.634,E2 -11650.634} C_VEL
LIN {X 0,Y 390.056,Z 422.896,A -85,B 0,C 180,E1 -11653.886,E2 -11653.886} C_VEL
LIN {X 0,Y 390.062,Z 422.901,A -85,B 0,C 180,E1 -11656.79,E2 -11656.79} C_VEL
LIN {X 0,Y 390.059,Z 422.899,A -85,B 0,C 180,E1 -11659.561,E2 -11659.561} C_VEL
LIN {X 0,Y 390.048,Z 422.899,A -85,B 0,C 180,E1 -11662.449,E2 -11662.449} C_VEL
LIN {X 0,Y 390.087,Z 422.897,A -85,B 0,C 180,E1 -11666.047,E2 -11666.047} C_VEL
LIN {X 0,Y 390.05,Z 422.901,A -85,B 0,C 180,E1 -11669.869,E2 -11669.869} C_VEL
LIN {X 0,Y 390.116,Z 422.888,A -85,B 0,C 180,E1 -11673.232,E2 -11673.232} C_VEL
LIN {X 0,Y 390.07,Z 422.894,A -85,B 0,C 180,E1 -11676.764,E2 -11676.764} C_VEL
LIN {X 0,Y 390.107,Z 422.894,A -85,B 0,C 180,E1 -11679.983,E2 -11679.983} C_VEL
LIN {X 0,Y 390.142,Z 422.886,A -85,B 0,C 180,E1 -11683.248,E2 -11683.248} C_VEL
LIN {X 0,Y 390.198,Z 422.878,A -85,B 0,C 180,E1 -11686.562,E2 -11686.562} C_VEL
LIN {X 0,Y 390.176,Z 422.885,A -85,B 0,C 180,E1 -11689.623,E2 -11689.623} C_VEL
LIN {X 0,Y 390.288,Z 422.866,A -85,B 0,C 180,E1 -11692.759,E2 -11692.759} C_VEL
LIN {X 0,Y 390.23,Z 422.874,A -85,B 0,C 180,E1 -11694.834,E2 -11694.834} C_VEL
LIN {X 0,Y 390.425,Z 422.853,A -85,B 0,C 180,E1 -11697.937,E2 -11697.937} C_VEL
LIN {X 0,Y 390.554,Z 422.836,A -85,B 0,C 180,E1 -11700,E2 -11700} C_VEL
LIN {X 0,Y 390.314,Z 422.865,A -85,B 0,C 180,E1 -11703.097,E2 -11703.097} C_VEL
LIN {X 0,Y 390.293,Z 422.866,A -85,B 0,C 180,E1 -11706.632,E2 -11706.632} C_VEL
LIN {X 0,Y 390.198,Z 422.882,A -85,B 0,C 180,E1 -11709.329,E2 -11709.329} C_VEL
LIN {X 0,Y 390.182,Z 422.88,A -85,B 0,C 180,E1 -11712.483,E2 -11712.483} C_VEL
LIN {X 0,Y 390.144,Z 422.888,A -85,B 0,C 180,E1 -11715.677,E2 -11715.677} C_VEL
LIN {X 0,Y 390.109,Z 422.891,A -85,B 0,C 180,E1 -11718.922,E2 -11718.922} C_VEL
LIN {X 0,Y 390.051,Z 422.896,A -85,B 0,C 180,E1 -11722.234,E2 -11722.234} C_VEL
LIN {X 0,Y 390.123,Z 422.889,A -85,B 0,C 180,E1 -11725.743,E2 -11725.743} C_VEL
LIN {X 0,Y 390.062,Z 422.9,A -85,B 0,C 180,E1 -11729.109,E2 -11729.109} C_VEL
LIN {X 0,Y 390.046,Z 422.898,A -85,B 0,C 180,E1 -11732.721,E2 -11732.721} C_VEL
LIN {X 0,Y 390.059,Z 422.896,A -85,B 0,C 180,E1 -11735.825,E2 -11735.825} C_VEL
LIN {X 0,Y 390.071,Z 422.899,A -85,B 0,C 180,E1 -11739.218,E2 -11739.218} C_VEL
LIN {X 0,Y 390.047,Z 422.897,A -85,B 0,C 180,E1 -11742.374,E2 -11742.374} C_VEL
LIN {X 0,Y 390.105,Z 422.889,A -85,B 0,C 180,E1 -11746.106,E2 -11746.106} C_VEL
LIN {X 0,Y 390.086,Z 422.897,A -85,B 0,C 180,E1 -11749.174,E2 -11749.174} C_VEL
LIN {X 0,Y 390.05,Z 422.898,A -85,B 0,C 180,E1 -11752.448,E2 -11752.448} C_VEL
LIN {X 0,Y 390.071,Z 422.894,A -85,B 0,C 180,E1 -11756.045,E2 -11756.045} C_VEL
LIN {X 0,Y 390.05,Z 422.896,A -85,B 0,C 180,E1 -11759.869,E2 -11759.869} C_VEL
LIN {X 0,Y 390.117,Z 422.89,A -85,B 0,C 180,E1 -11763.232,E2 -11763.232} C_VEL
LIN {X 0,Y 390.11,Z 422.894,A -85,B 0,C 180,E1 -11766.75,E2 -11766.75} C_VEL
LIN {X 0,Y 390.107,Z 422.889,A -85,B 0,C 180,E1 -11769.983,E2 -11769.983} C_VEL
LIN {X 0,Y 390.134,Z 422.891,A -85,B 0,C 180,E1 -11772.308,E2 -11772.308} C_VEL
LIN {X 0,Y 393.991,Z 435.166,A -85,B 0,C 180,E1 -11773.283,E2 -11773.283} C_VEL
LIN {X 0,Y 395.596,Z 440.96,A -85,B 0,C 180,E1 -11773.821,E2 -11773.821} C_VEL
LIN {X 0,Y 394.886,Z 451.663,A -85,B 0,C 180,E1 -11774.781,E2 -11774.781} C_VEL
LIN {X 0,Y 394.107,Z 461.993,A -85,B 0,C 180,E1 -11775.938,E2 -11775.938} C_VEL
LIN {X 0,Y 393.432,Z 470.414,A -85,B 0,C 180,E1 -11777.097,E2 -11777.097} C_VEL
LIN {X 0,Y 392.704,Z 478.166,A -85,B 0,C 180,E1 -11778.385,E2 -11778.385} C_VEL
LIN {X 0,Y 391.905,Z 485.742,A -85,B 0,C 180,E1 -11779.93,E2 -11779.93} C_VEL
LIN {X 0,Y 391.451,Z 491.011,A -85,B 0,C 180,E1 -11781.258,E2 -11781.258} C_VEL
LIN {X 0,Y 391.064,Z 495.86,A -85,B 0,C 180,E1 -11782.773,E2 -11782.773} C_VEL
LIN {X 0,Y 390.556,Z 499.75,A -85,B 0,C 180,E1 -11784.32,E2 -11784.32} C_VEL
LIN {X 0,Y 390.209,Z 502.615,A -85,B 0,C 180,E1 -11785.869,E2 -11785.869} C_VEL
LIN {X 0,Y 390.029,Z 503.991,A -85,B 0,C 180,E1 -11786.901,E2 -11786.901} C_VEL
LIN {X 0,Y 390.033,Z 505.54,A -85,B 0,C 180,E1 -11788.967,E2 -11788.967} C_VEL
LIN {X 0,Y 390.063,Z 505.762,A -85,B 0,C 180,E1 -11790,E2 -11790} C_VEL
LIN {X 0,Y 390.033,Z 505.021,A -85,B 0,C 180,E1 -11792.065,E2 -11792.065} C_VEL
LIN {X 0,Y 390.023,Z 504.092,A -85,B 0,C 180,E1 -11793.099,E2 -11793.099} C_VEL
LIN {X 0,Y 390.199,Z 502.762,A -85,B 0,C 180,E1 -11794.131,E2 -11794.131} C_VEL
LIN {X 0,Y 390.55,Z 499.949,A -85,B 0,C 180,E1 -11795.68,E2 -11795.68} C_VEL
LIN {X 0,Y 391.033,Z 496.131,A -85,B 0,C 180,E1 -11797.227,E2 -11797.227} C_VEL
LIN {X 0,Y 391.413,Z 490.257,A -85,B 0,C 180,E1 -11799.049,E2 -11799.049} C_VEL
LIN {X 0,Y 392.145,Z 483.835,A -85,B 0,C 180,E1 -11800.585,E2 -11800.585} C_VEL
LIN {X 0,Y 392.973,Z 475.807,A -85,B 0,C 180,E1 -11802.13,E2 -11802.13} C_VEL
LIN {X 0,Y 393.635,Z 467.59,A -85,B 0,C 180,E1 -11803.421,E2 -11803.421} C_VEL
LIN {X 0,Y 394.454,Z 457.404,A -85,B 0,C 180,E1 -11804.708,E2 -11804.708} C_VEL
LIN {X 0,Y 395.285,Z 446.384,A -85,B 0,C 180,E1 -11805.817,E2 -11805.817} C_VEL
LIN {X 0,Y 395.46,Z 440.486,A -85,B 0,C 180,E1 -11806.326,E2 -11806.326} C_VEL
LIN {X 0,Y 392.361,Z 429.784,A -85,B 0,C 180,E1 -11807.27,E2 -11807.27} C_VEL
LIN {X 0,Y 390.131,Z 422.891,A -85,B 0,C 180,E1 -11807.793,E2 -11807.793} C_VEL
LIN {X 0,Y 390.056,Z 422.899,A -85,B 0,C 180,E1 -11811.152,E2 -11811.152} C_VEL
LIN {X 0,Y 389.349,Z 422.985,A -85,B 0,C 180,E1 -11812.013,E2 -11812.013} C_VEL
LIN {X 0,Y 386.49,Z 423.345,A -85,B 0,C 180,E1 -11813.415,E2 -11813.415} C_VEL
LIN {X 0,Y 384.116,Z 423.638,A -85,B 0,C 180,E1 -11814.547,E2 -11814.547} C_VEL
LIN {X 0,Y 383.129,Z 423.763,A -85,B 0,C 180,E1 -11815.423,E2 -11815.423} C_VEL
LIN {X 0,Y 383.064,Z 423.766,A -85,B 0,C 180,E1 -11815.719,E2 -11815.719} C_VEL
LIN {X 0,Y 383.02,Z 423.772,A -85,B 0,C 180,E1 -11818.494,E2 -11818.494} C_VEL
LIN {X 0,Y 383.012,Z 423.772,A -85,B 0,C 180,E1 -11822.15,E2 -11822.15} C_VEL
LIN {X 0,Y 383.021,Z 423.773,A -85,B 0,C 180,E1 -11824.668,E2 -11824.668} C_VEL
LIN {X 0,Y 383.006,Z 423.774,A -85,B 0,C 180,E1 -11827.905,E2 -11827.905} C_VEL
LIN {X 0,Y 383.049,Z 423.772,A -85,B 0,C 180,E1 -11831.339,E2 -11831.339} C_VEL
LIN {X 0,Y 383.039,Z 423.77,A -85,B 0,C 180,E1 -11834.31,E2 -11834.31} C_VEL
LIN {X 0,Y 383.012,Z 423.776,A -85,B 0,C 180,E1 -11837.24,E2 -11837.24} C_VEL
LIN {X 0,Y 383.017,Z 423.773,A -85,B 0,C 180,E1 -11840.413,E2 -11840.413} C_VEL
LIN {X 0,Y 383.027,Z 423.771,A -85,B 0,C 180,E1 -11844.044,E2 -11844.044} C_VEL
LIN {X 0,Y 382.989,Z 423.776,A -85,B 0,C 180,E1 -11847.578,E2 -11847.578} C_VEL
LIN {X 0,Y 382.994,Z 423.776,A -85,B 0,C 180,E1 -11850.3,E2 -11850.3} C_VEL
LIN {X 0,Y 383.082,Z 423.764,A -85,B 0,C 180,E1 -11854.021,E2 -11854.021} C_VEL
LIN {X 0,Y 383.01,Z 423.774,A -85,B 0,C 180,E1 -11857.335,E2 -11857.335} C_VEL
LIN {X 0,Y 383.063,Z 423.772,A -85,B 0,C 180,E1 -11860.716,E2 -11860.716} C_VEL
LIN {X 0,Y 383.084,Z 423.765,A -85,B 0,C 180,E1 -11864.027,E2 -11864.027} C_VEL
LIN {X 0,Y 383.144,Z 423.757,A -85,B 0,C 180,E1 -11867.284,E2 -11867.284} C_VEL
LIN {X 0,Y 383.148,Z 423.761,A -85,B 0,C 180,E1 -11870.498,E2 -11870.498} C_VEL
LIN {X 0,Y 383.278,Z 423.74,A -85,B 0,C 180,E1 -11873.683,E2 -11873.683} C_VEL
LIN {X 0,Y 383.391,Z 423.727,A -85,B 0,C 180,E1 -11877.899,E2 -11877.899} C_VEL
LIN {X 0,Y 383.523,Z 423.711,A -85,B 0,C 180,E1 -11880,E2 -11880} C_VEL
LIN {X 0,Y 383.255,Z 423.743,A -85,B 0,C 180,E1 -11883.154,E2 -11883.154} C_VEL
LIN {X 0,Y 383.279,Z 423.745,A -85,B 0,C 180,E1 -11886.316,E2 -11886.316} C_VEL
LIN {X 0,Y 383.147,Z 423.756,A -85,B 0,C 180,E1 -11889.502,E2 -11889.502} C_VEL
LIN {X 0,Y 383.143,Z 423.758,A -85,B 0,C 180,E1 -11892.716,E2 -11892.716} C_VEL
LIN {X 0,Y 383.084,Z 423.768,A -85,B 0,C 180,E1 -11895.973,E2 -11895.973} C_VEL
LIN {X 0,Y 383.063,Z 423.766,A -85,B 0,C 180,E1 -11899.284,E2 -11899.284} C_VEL
LIN {X 0,Y 382.993,Z 423.776,A -85,B 0,C 180,E1 -11902.666,E2 -11902.666} C_VEL
LIN {X 0,Y 383.081,Z 423.77,A -85,B 0,C 180,E1 -11906.123,E2 -11906.123} C_VEL
LIN {X 0,Y 383.019,Z 423.774,A -85,B 0,C 180,E1 -11908.494,E2 -11908.494} C_VEL
LIN {X 0,Y 383.012,Z 423.778,A -85,B 0,C 180,E1 -11912.15,E2 -11912.15} C_VEL
LIN {X 0,Y 383.02,Z 423.772,A -85,B 0,C 180,E1 -11914.668,E2 -11914.668} C_VEL
LIN {X 0,Y 383.003,Z 423.779,A -85,B 0,C 180,E1 -11917.904,E2 -11917.904} C_VEL
LIN {X 0,Y 382.986,Z 423.777,A -85,B 0,C 180,E1 -11921.347,E2 -11921.347} C_VEL
LIN {X 0,Y 383,Z 423.78,A -85,B 0,C 180,E1 -11924.304,E2 -11924.304} C_VEL
LIN {X 0,Y 383.02,Z 423.932,A -85,B 0,C 180,E1 -11925.792,E2 -11925.792} C_VEL
LIN {X 0,Y 385.049,Z 433.474,A -85,B 0,C 180,E1 -11929.356,E2 -11929.356} C_VEL
LIN {X 0,Y 386.618,Z 442.518,A -85,B 0,C 180,E1 -11932.486,E2 -11932.486} C_VEL
LIN {X 0,Y 386.202,Z 448.54,A -85,B 0,C 180,E1 -11934.386,E2 -11934.386} C_VEL
LIN {X 0,Y 385.207,Z 460.554,A -85,B 0,C 180,E1 -11938.055,E2 -11938.055} C_VEL
LIN {X 0,Y 384.13,Z 474.451,A -85,B 0,C 180,E1 -11942.19,E2 -11942.19} C_VEL
LIN {X 0,Y 383.383,Z 486.174,A -85,B 0,C 180,E1 -11945.641,E2 -11945.641} C_VEL
LIN {X 0,Y 382.756,Z 499.56,A -85,B 0,C 180,E1 -11949.582,E2 -11949.582} C_VEL
LIN {X 0,Y 382.568,Z 504.352,A -85,B 0,C 180,E1 -11951.004,E2 -11951.004} C_VEL
LIN {X 0,Y 384.465,Z 520.343,A -85,B 0,C 180,E1 -11951.609,E2 -11951.609} C_VEL
LIN {X 0,Y 385.394,Z 532.825,A -85,B 0,C 180,E1 -11952.268,E2 -11952.268} C_VEL
LIN {X 0,Y 385.894,Z 546.231,A -85,B 0,C 180,E1 -11953.195,E2 -11953.195} C_VEL
LIN {X 0,Y 385.768,Z 552.754,A -85,B 0,C 180,E1 -11953.734,E2 -11953.734} C_VEL
LIN {X 0,Y 384.792,Z 563.502,A -85,B 0,C 180,E1 -11954.779,E2 -11954.779} C_VEL
LIN {X 0,Y 383.868,Z 573.734,A -85,B 0,C 180,E1 -11956.012,E2 -11956.012} C_VEL
LIN {X 0,Y 383.245,Z 582.386,A -85,B 0,C 180,E1 -11957.288,E2 -11957.288} C_VEL
LIN {X 0,Y 382.602,Z 591.217,A -85,B 0,C 180,E1 -11958.879,E2 -11958.879} C_VEL
LIN {X 0,Y 382.304,Z 598.321,A -85,B 0,C 180,E1 -11960.477,E2 -11960.477} C_VEL
LIN {X 0,Y 382.15,Z 604.036,A -85,B 0,C 180,E1 -11962.072,E2 -11962.072} C_VEL
LIN {X 0,Y 382.217,Z 608.551,A -85,B 0,C 180,E1 -11963.666,E2 -11963.666} C_VEL
LIN {X 0,Y 382.27,Z 610.944,A -85,B 0,C 180,E1 -11964.726,E2 -11964.726} C_VEL
LIN {X 0,Y 382.44,Z 612.904,A -85,B 0,C 180,E1 -11965.785,E2 -11965.785} C_VEL
LIN {X 0,Y 382.438,Z 614.356,A -85,B 0,C 180,E1 -11966.84,E2 -11966.84} C_VEL
LIN {X 0,Y 382.475,Z 615.397,A -85,B 0,C 180,E1 -11967.894,E2 -11967.894} C_VEL
LIN {X 0,Y 382.762,Z 616.293,A -85,B 0,C 180,E1 -11970,E2 -11970} C_VEL
LIN {X 0,Y 382.476,Z 615.394,A -85,B 0,C 180,E1 -11972.106,E2 -11972.106} C_VEL
LIN {X 0,Y 382.439,Z 614.353,A -85,B 0,C 180,E1 -11973.16,E2 -11973.16} C_VEL
LIN {X 0,Y 382.44,Z 612.898,A -85,B 0,C 180,E1 -11974.216,E2 -11974.216} C_VEL
LIN {X 0,Y 382.208,Z 609.811,A -85,B 0,C 180,E1 -11975.805,E2 -11975.805} C_VEL
LIN {X 0,Y 382.143,Z 605.67,A -85,B 0,C 180,E1 -11977.397,E2 -11977.397} C_VEL
LIN {X 0,Y 382.232,Z 599.334,A -85,B 0,C 180,E1 -11979.258,E2 -11979.258} C_VEL
LIN {X 0,Y 382.525,Z 592.453,A -85,B 0,C 180,E1 -11980.855,E2 -11980.855} C_VEL
LIN {X 0,Y 383.057,Z 583.959,A -85,B 0,C 180,E1 -11982.45,E2 -11982.45} C_VEL
LIN {X 0,Y 383.606,Z 577.128,A -85,B 0,C 180,E1 -11983.509,E2 -11983.509} C_VEL
LIN {X 0,Y 384.515,Z 566.984,A -85,B 0,C 180,E1 -11984.826,E2 -11984.826} C_VEL
LIN {X 0,Y 385.364,Z 556.995,A -85,B 0,C 180,E1 -11985.876,E2 -11985.876} C_VEL
LIN {X 0,Y 385.972,Z 547.877,A -85,B 0,C 180,E1 -11986.666,E2 -11986.666} C_VEL
LIN {X 0,Y 385.523,Z 536.109,A -85,B 0,C 180,E1 -11987.522,E2 -11987.522} C_VEL
LIN {X 0,Y 384.641,Z 522.401,A -85,B 0,C 180,E1 -11988.283,E2 -11988.283} C_VEL
LIN {X 0,Y 383.095,Z 508.734,A -85,B 0,C 180,E1 -11988.837,E2 -11988.837} C_VEL
LIN {X 0,Y 382.57,Z 504.42,A -85,B 0,C 180,E1 -11988.965,E2 -11988.965} C_VEL
LIN {X 0,Y 383.174,Z 490.448,A -85,B 0,C 180,E1 -11993.096,E2 -11993.096} C_VEL
LIN {X 0,Y 383.858,Z 478.343,A -85,B 0,C 180,E1 -11996.655,E2 -11996.655} C_VEL
LIN {X 0,Y 384.666,Z 466.477,A -85,B 0,C 180,E1 -12000.162,E2 -12000.162} C_VEL
LIN {X 0,Y 385.551,Z 455.494,A -85,B 0,C 180,E1 -12003.464,E2 -12003.464} C_VEL
LIN {X 0,Y 386.619,Z 444.417,A -85,B 0,C 180,E1 -12006.885,E2 -12006.885} C_VEL
LIN {X 0,Y 386.3,Z 440.4,A -85,B 0,C 180,E1 -12008.212,E2 -12008.212} C_VEL
LIN {X 0,Y 384.742,Z 432.122,A -85,B 0,C 180,E1 -12011.118,E2 -12011.118} C_VEL
LIN {X 0,Y 382.998,Z 423.778,A -85,B 0,C 180,E1 -12014.304,E2 -12014.304} C_VEL
LIN {X 0,Y 383.012,Z 423.777,A -85,B 0,C 180,E1 -12017.24,E2 -12017.24} C_VEL
LIN {X 0,Y 383.018,Z 423.775,A -85,B 0,C 180,E1 -12020.413,E2 -12020.413} C_VEL
LIN {X 0,Y 383.029,Z 423.776,A -85,B 0,C 180,E1 -12024.045,E2 -12024.045} C_VEL
LIN {X 0,Y 382.99,Z 423.777,A -85,B 0,C 180,E1 -12027.578,E2 -12027.578} C_VEL
LIN {X 0,Y 382.995,Z 423.778,A -85,B 0,C 180,E1 -12030.3,E2 -12030.3} C_VEL
LIN {X 0,Y 383.083,Z 423.769,A -85,B 0,C 180,E1 -12034.021,E2 -12034.021} C_VEL
LIN {X 0,Y 382.994,Z 423.776,A -85,B 0,C 180,E1 -12037.334,E2 -12037.334} C_VEL
LIN {X 0,Y 383.064,Z 423.766,A -85,B 0,C 180,E1 -12040.716,E2 -12040.716} C_VEL
LIN {X 0,Y 383.085,Z 423.768,A -85,B 0,C 180,E1 -12044.027,E2 -12044.027} C_VEL
LIN {X 0,Y 383.145,Z 423.758,A -85,B 0,C 180,E1 -12047.284,E2 -12047.284} C_VEL
LIN {X 0,Y 383.148,Z 423.756,A -85,B 0,C 180,E1 -12050.498,E2 -12050.498} C_VEL
LIN {X 0,Y 383.28,Z 423.745,A -85,B 0,C 180,E1 -12053.684,E2 -12053.684} C_VEL
LIN {X 0,Y 383.392,Z 423.729,A -85,B 0,C 180,E1 -12057.899,E2 -12057.899} C_VEL
LIN {X 0,Y 383.524,Z 423.711,A -85,B 0,C 180,E1 -12060,E2 -12060} C_VEL
LIN {X 0,Y 383.251,Z 423.745,A -85,B 0,C 180,E1 -12063.154,E2 -12063.154} C_VEL
LIN {X 0,Y 383.253,Z 423.743,A -85,B 0,C 180,E1 -12066.622,E2 -12066.622} C_VEL
LIN {X 0,Y 383.149,Z 423.761,A -85,B 0,C 180,E1 -12069.502,E2 -12069.502} C_VEL
LIN {X 0,Y 383.145,Z 423.756,A -85,B 0,C 180,E1 -12072.716,E2 -12072.716} C_VEL
LIN {X 0,Y 383.085,Z 423.765,A -85,B 0,C 180,E1 -12075.973,E2 -12075.973} C_VEL
LIN {X 0,Y 383.064,Z 423.771,A -85,B 0,C 180,E1 -12079.284,E2 -12079.284} C_VEL
LIN {X 0,Y 383.016,Z 423.773,A -85,B 0,C 180,E1 -12082.664,E2 -12082.664} C_VEL
LIN {X 0,Y 383.083,Z 423.764,A -85,B 0,C 180,E1 -12086.123,E2 -12086.123} C_VEL
LIN {X 0,Y 382.995,Z 423.777,A -85,B 0,C 180,E1 -12089.7,E2 -12089.7} C_VEL
LIN {X 0,Y 383.006,Z 423.778,A -85,B 0,C 180,E1 -12093.401,E2 -12093.401} C_VEL
LIN {X 0,Y 383.035,Z 423.77,A -85,B 0,C 180,E1 -12096.165,E2 -12096.165} C_VEL
LIN {X 0,Y 383.011,Z 423.773,A -85,B 0,C 180,E1 -12099.958,E2 -12099.958} C_VEL
LIN {X 0,Y 383.008,Z 423.776,A -85,B 0,C 180,E1 -12102.779,E2 -12102.779} C_VEL
LIN {X 0,Y 383.042,Z 423.769,A -85,B 0,C 180,E1 -12105.795,E2 -12105.795} C_VEL
LIN {X 0,Y 383.047,Z 423.772,A -85,B 0,C 180,E1 -12108.786,E2 -12108.786} C_VEL
LIN {X 0,Y 383.007,Z 423.773,A -85,B 0,C 180,E1 -12112.095,E2 -12112.095} C_VEL
LIN {X 0,Y 383.021,Z 423.774,A -85,B 0,C 180,E1 -12115.332,E2 -12115.332} C_VEL
LIN {X 0,Y 382.986,Z 423.78,A -85,B 0,C 180,E1 -12119.081,E2 -12119.081} C_VEL
LIN {X 0,Y 383.06,Z 423.772,A -85,B 0,C 180,E1 -12122.698,E2 -12122.698} C_VEL
LIN {X 0,Y 383.055,Z 423.771,A -85,B 0,C 180,E1 -12125.04,E2 -12125.04} C_VEL
LIN {X 0,Y 382.996,Z 423.778,A -85,B 0,C 180,E1 -12128.469,E2 -12128.469} C_VEL
LIN {X 0,Y 383.097,Z 423.851,A -85,B 0,C 180,E1 -12131.969,E2 -12131.969} C_VEL
LIN {X 0,Y 387.064,Z 436.208,A -85,B 0,C 180,E1 -12132.975,E2 -12132.975} C_VEL
LIN {X 0,Y 388.741,Z 442.221,A -85,B 0,C 180,E1 -12133.548,E2 -12133.548} C_VEL
LIN {X 0,Y 388.116,Z 452.672,A -85,B 0,C 180,E1 -12134.508,E2 -12134.508} C_VEL
LIN {X 0,Y 387.295,Z 463.002,A -85,B 0,C 180,E1 -12135.685,E2 -12135.685} C_VEL
LIN {X 0,Y 386.586,Z 471.423,A -85,B 0,C 180,E1 -12136.865,E2 -12136.865} C_VEL
LIN {X 0,Y 385.826,Z 479.174,A -85,B 0,C 180,E1 -12138.175,E2 -12138.175} C_VEL
LIN {X 0,Y 384.988,Z 486.749,A -85,B 0,C 180,E1 -12139.747,E2 -12139.747} C_VEL
LIN {X 0,Y 384.506,Z 492.018,A -85,B 0,C 180,E1 -12141.099,E2 -12141.099} C_VEL
LIN {X 0,Y 384.095,Z 496.867,A -85,B 0,C 180,E1 -12142.641,E2 -12142.641} C_VEL
LIN {X 0,Y 383.566,Z 500.755,A -85,B 0,C 180,E1 -12144.216,E2 -12144.216} C_VEL
LIN {X 0,Y 383.199,Z 503.621,A -85,B 0,C 180,E1 -12145.793,E2 -12145.793} C_VEL
LIN {X 0,Y 383.011,Z 504.997,A -85,B 0,C 180,E1 -12146.844,E2 -12146.844} C_VEL
LIN {X 0,Y 383.023,Z 506.543,A -85,B 0,C 180,E1 -12148.949,E2 -12148.949} C_VEL
LIN {X 0,Y 383.046,Z 506.766,A -85,B 0,C 180,E1 -12150,E2 -12150} C_VEL
LIN {X 0,Y 383.011,Z 506.026,A -85,B 0,C 180,E1 -12152.103,E2 -12152.103} C_VEL
LIN {X 0,Y 383.005,Z 505.097,A -85,B 0,C 180,E1 -12153.156,E2 -12153.156} C_VEL
LIN {X 0,Y 383.189,Z 503.766,A -85,B 0,C 180,E1 -12154.207,E2 -12154.207} C_VEL
LIN {X 0,Y 383.56,Z 500.953,A -85,B 0,C 180,E1 -12155.784,E2 -12155.784} C_VEL
LIN {X 0,Y 384.062,Z 497.135,A -85,B 0,C 180,E1 -12157.359,E2 -12157.359} C_VEL
LIN {X 0,Y 384.484,Z 491.226,A -85,B 0,C 180,E1 -12159.222,E2 -12159.222} C_VEL
LIN {X 0,Y 385.239,Z 484.838,A -85,B 0,C 180,E1 -12160.777,E2 -12160.777} C_VEL
LIN {X 0,Y 386.115,Z 476.808,A -85,B 0,C 180,E1 -12162.349,E2 -12162.349} C_VEL
LIN {X 0,Y 386.802,Z 468.592,A -85,B 0,C 180,E1 -12163.663,E2 -12163.663} C_VEL
LIN {X 0,Y 387.66,Z 458.405,A -85,B 0,C 180,E1 -12164.972,E2 -12164.972} C_VEL
LIN {X 0,Y 388.505,Z 447.762,A -85,B 0,C 180,E1 -12166.065,E2 -12166.065} C_VEL
LIN {X 0,Y 388.648,Z 441.944,A -85,B 0,C 180,E1 -12166.582,E2 -12166.582} C_VEL
LIN {X 0,Y 385.434,Z 431.132,A -85,B 0,C 180,E1 -12167.571,E2 -12167.571} C_VEL
LIN {X 0,Y 383.091,Z 423.768,A -85,B 0,C 180,E1 -12168.172,E2 -12168.172} C_VEL
LIN {X 0,Y 382.996,Z 423.779,A -85,B 0,C 180,E1 -12171.531,E2 -12171.531} C_VEL
LIN {X 0,Y 383.055,Z 423.771,A -85,B 0,C 180,E1 -12174.96,E2 -12174.96} C_VEL
LIN {X 0,Y 383.064,Z 423.766,A -85,B 0,C 180,E1 -12175.719,E2 -12175.719} C_VEL
LIN {X 0,Y 382.435,Z 423.847,A -85,B 0,C 180,E1 -12176.597,E2 -12176.597} C_VEL
LIN {X 0,Y 379.579,Z 424.2,A -85,B 0,C 180,E1 -12178.023,E2 -12178.023} C_VEL
LIN {X 0,Y 377.126,Z 424.511,A -85,B 0,C 180,E1 -12179.176,E2 -12179.176} C_VEL
LIN {X 0,Y 376.058,Z 424.639,A -85,B 0,C 180,E1 -12180.068,E2 -12180.068} C_VEL
LIN {X 0,Y 375.965,Z 424.65,A -85,B 0,C 180,E1 -12180.371,E2 -12180.371} C_VEL
LIN {X 0,Y 375.964,Z 424.65,A -85,B 0,C 180,E1 -12184.111,E2 -12184.111} C_VEL
LIN {X 0,Y 375.958,Z 424.654,A -85,B 0,C 180,E1 -12186.741,E2 -12186.741} C_VEL
LIN {X 0,Y 376.002,Z 424.646,A -85,B 0,C 180,E1 -12189.973,E2 -12189.973} C_VEL
LIN {X 0,Y 375.992,Z 424.651,A -85,B 0,C 180,E1 -12193.198,E2 -12193.198} C_VEL
LIN {X 0,Y 375.94,Z 424.658,A -85,B 0,C 180,E1 -12196.81,E2 -12196.81} C_VEL
LIN {X 0,Y 375.965,Z 424.653,A -85,B 0,C 180,E1 -12200.537,E2 -12200.537} C_VEL
LIN {X 0,Y 375.966,Z 424.651,A -85,B 0,C 180,E1 -12203.495,E2 -12203.495} C_VEL
LIN {X 0,Y 375.962,Z 424.651,A -85,B 0,C 180,E1 -12205.889,E2 -12205.889} C_VEL
LIN {X 0,Y 375.967,Z 424.65,A -85,B 0,C 180,E1 -12209.687,E2 -12209.687} C_VEL
LIN {X 0,Y 376.022,Z 424.644,A -85,B 0,C 180,E1 -12213.348,E2 -12213.348} C_VEL
LIN {X 0,Y 375.998,Z 424.651,A -85,B 0,C 180,E1 -12216.888,E2 -12216.888} C_VEL
LIN {X 0,Y 376,Z 424.649,A -85,B 0,C 180,E1 -12220.339,E2 -12220.339} C_VEL
LIN {X 0,Y 376.032,Z 424.642,A -85,B 0,C 180,E1 -12223.719,E2 -12223.719} C_VEL
LIN {X 0,Y 376.109,Z 424.634,A -85,B 0,C 180,E1 -12227.042,E2 -12227.042} C_VEL
LIN {X 0,Y 376.118,Z 424.635,A -85,B 0,C 180,E1 -12230.318,E2 -12230.318} C_VEL
LIN {X 0,Y 376.235,Z 424.617,A -85,B 0,C 180,E1 -12233.565,E2 -12233.565} C_VEL
LIN {X 0,Y 376.357,Z 424.602,A -85,B 0,C 180,E1 -12237.86,E2 -12237.86} C_VEL
LIN {X 0,Y 376.492,Z 424.587,A -85,B 0,C 180,E1 -12240,E2 -12240} C_VEL
LIN {X 0,Y 376.193,Z 424.622,A -85,B 0,C 180,E1 -12243.213,E2 -12243.213} C_VEL
LIN {X 0,Y 376.235,Z 424.622,A -85,B 0,C 180,E1 -12246.435,E2 -12246.435} C_VEL
LIN {X 0,Y 376.117,Z 424.632,A -85,B 0,C 180,E1 -12249.681,E2 -12249.681} C_VEL
LIN {X 0,Y 376.092,Z 424.635,A -85,B 0,C 180,E1 -12253.658,E2 -12253.658} C_VEL
LIN {X 0,Y 376.046,Z 424.641,A -85,B 0,C 180,E1 -12257.607,E2 -12257.607} C_VEL
LIN {X 0,Y 375.98,Z 424.649,A -85,B 0,C 180,E1 -12260.832,E2 -12260.832} C_VEL
LIN {X 0,Y 375.99,Z 424.652,A -85,B 0,C 180,E1 -12264.282,E2 -12264.282} C_VEL
LIN {X 0,Y 376.021,Z 424.644,A -85,B 0,C 180,E1 -12266.652,E2 -12266.652} C_VEL
LIN {X 0,Y 375.966,Z 424.653,A -85,B 0,C 180,E1 -12270.313,E2 -12270.313} C_VEL
LIN {X 0,Y 375.964,Z 424.655,A -85,B 0,C 180,E1 -12274.111,E2 -12274.111} C_VEL
LIN {X 0,Y 375.957,Z 424.651,A -85,B 0,C 180,E1 -12276.741,E2 -12276.741} C_VEL
LIN {X 0,Y 375.991,Z 424.653,A -85,B 0,C 180,E1 -12279.971,E2 -12279.971} C_VEL
LIN {X 0,Y 375.933,Z 424.66,A -85,B 0,C 180,E1 -12283.766,E2 -12283.766} C_VEL
LIN {X 0,Y 375.949,Z 424.727,A -85,B 0,C 180,E1 -12285.361,E2 -12285.361} C_VEL
LIN {X 0,Y 377.813,Z 433.655,A -85,B 0,C 180,E1 -12288.785,E2 -12288.785} C_VEL
LIN {X 0,Y 379.386,Z 441.926,A -85,B 0,C 180,E1 -12291.75,E2 -12291.75} C_VEL
LIN {X 0,Y 379.654,Z 444.886,A -85,B 0,C 180,E1 -12292.75,E2 -12292.75} C_VEL
LIN {X 0,Y 378.662,Z 455.664,A -85,B 0,C 180,E1 -12296.165,E2 -12296.165} C_VEL
LIN {X 0,Y 377.923,Z 464.219,A -85,B 0,C 180,E1 -12298.808,E2 -12298.808} C_VEL
LIN {X 0,Y 376.93,Z 477.429,A -85,B 0,C 180,E1 -12302.818,E2 -12302.818} C_VEL
LIN {X 0,Y 376.162,Z 489.91,A -85,B 0,C 180,E1 -12306.575,E2 -12306.575} C_VEL
LIN {X 0,Y 375.531,Z 503.317,A -85,B 0,C 180,E1 -12310.634,E2 -12310.634} C_VEL
LIN {X 0,Y 377.413,Z 519.288,A -85,B 0,C 180,E1 -12311.253,E2 -12311.253} C_VEL
LIN {X 0,Y 378.473,Z 532.688,A -85,B 0,C 180,E1 -12311.988,E2 -12311.988} C_VEL
LIN {X 0,Y 378.874,Z 545.187,A -85,B 0,C 180,E1 -12312.874,E2 -12312.874} C_VEL
LIN {X 0,Y 378.928,Z 551.738,A -85,B 0,C 180,E1 -12313.432,E2 -12313.432} C_VEL
LIN {X 0,Y 377.835,Z 562.473,A -85,B 0,C 180,E1 -12314.491,E2 -12314.491} C_VEL
LIN {X 0,Y 376.943,Z 572.716,A -85,B 0,C 180,E1 -12315.75,E2 -12315.75} C_VEL
LIN {X 0,Y 376.296,Z 581.369,A -85,B 0,C 180,E1 -12317.049,E2 -12317.049} C_VEL
LIN {X 0,Y 375.59,Z 590.196,A -85,B 0,C 180,E1 -12318.669,E2 -12318.669} C_VEL
LIN {X 0,Y 375.214,Z 597.294,A -85,B 0,C 180,E1 -12320.295,E2 -12320.295} C_VEL
LIN {X 0,Y 375.086,Z 603.017,A -85,B 0,C 180,E1 -12321.922,E2 -12321.922} C_VEL
LIN {X 0,Y 375.132,Z 607.532,A -85,B 0,C 180,E1 -12323.546,E2 -12323.546} C_VEL
LIN {X 0,Y 375.193,Z 609.929,A -85,B 0,C 180,E1 -12324.626,E2 -12324.626} C_VEL
LIN {X 0,Y 375.365,Z 611.89,A -85,B 0,C 180,E1 -12325.705,E2 -12325.705} C_VEL
LIN {X 0,Y 375.392,Z 613.347,A -85,B 0,C 180,E1 -12326.78,E2 -12326.78} C_VEL
LIN {X 0,Y 375.435,Z 614.39,A -85,B 0,C 180,E1 -12327.854,E2 -12327.854} C_VEL
LIN {X 0,Y 375.735,Z 615.288,A -85,B 0,C 180,E1 -12330,E2 -12330} C_VEL
LIN {X 0,Y 375.436,Z 614.386,A -85,B 0,C 180,E1 -12332.146,E2 -12332.146} C_VEL
LIN {X 0,Y 375.393,Z 613.343,A -85,B 0,C 180,E1 -12333.22,E2 -12333.22} C_VEL
LIN {X 0,Y 375.365,Z 611.883,A -85,B 0,C 180,E1 -12334.295,E2 -12334.295} C_VEL
LIN {X 0,Y 375.149,Z 608.795,A -85,B 0,C 180,E1 -12335.914,E2 -12335.914} C_VEL
LIN {X 0,Y 375.068,Z 604.649,A -85,B 0,C 180,E1 -12337.537,E2 -12337.537} C_VEL
LIN {X 0,Y 375.187,Z 598.311,A -85,B 0,C 180,E1 -12339.434,E2 -12339.434} C_VEL
LIN {X 0,Y 375.482,Z 591.425,A -85,B 0,C 180,E1 -12341.061,E2 -12341.061} C_VEL
LIN {X 0,Y 376.091,Z 582.936,A -85,B 0,C 180,E1 -12342.684,E2 -12342.684} C_VEL
LIN {X 0,Y 376.791,Z 573.857,A -85,B 0,C 180,E1 -12344.089,E2 -12344.089} C_VEL
LIN {X 0,Y 377.781,Z 563.598,A -85,B 0,C 180,E1 -12345.373,E2 -12345.373} C_VEL
LIN {X 0,Y 378.74,Z 553.083,A -85,B 0,C 180,E1 -12346.438,E2 -12346.438} C_VEL
LIN {X 0,Y 378.997,Z 548.451,A -85,B 0,C 180,E1 -12346.843,E2 -12346.843} C_VEL
LIN {X 0,Y 378.618,Z 537.199,A -85,B 0,C 180,E1 -12347.71,E2 -12347.71} C_VEL
LIN {X 0,Y 377.916,Z 524.447,A -85,B 0,C 180,E1 -12348.48,E2 -12348.48} C_VEL
LIN {X 0,Y 376.476,Z 510.734,A -85,B 0,C 180,E1 -12349.089,E2 -12349.089} C_VEL
LIN {X 0,Y 375.539,Z 503.341,A -85,B 0,C 180,E1 -12349.344,E2 -12349.344} C_VEL
LIN {X 0,Y 376.222,Z 488.801,A -85,B 0,C 180,E1 -12353.745,E2 -12353.745} C_VEL
LIN {X 0,Y 376.891,Z 477.392,A -85,B 0,C 180,E1 -12357.185,E2 -12357.185} C_VEL
LIN {X 0,Y 377.762,Z 465.854,A -85,B 0,C 180,E1 -12360.678,E2 -12360.678} C_VEL
LIN {X 0,Y 378.648,Z 455.611,A -85,B 0,C 180,E1 -12363.837,E2 -12363.837} C_VEL
LIN {X 0,Y 379.578,Z 446.234,A -85,B 0,C 180,E1 -12366.793,E2 -12366.793} C_VEL
LIN {X 0,Y 379.374,Z 441.878,A -85,B 0,C 180,E1 -12368.251,E2 -12368.251} C_VEL
LIN {X 0,Y 377.802,Z 433.598,A -85,B 0,C 180,E1 -12371.215,E2 -12371.215} C_VEL
LIN {X 0,Y 375.936,Z 424.659,A -85,B 0,C 180,E1 -12374.685,E2 -12374.685} C_VEL
LIN {X 0,Y 375.938,Z 424.659,A -85,B 0,C 180,E1 -12378.399,E2 -12378.399} C_VEL
LIN {X 0,Y 375.978,Z 424.651,A -85,B 0,C 180,E1 -12381.729,E2 -12381.729} C_VEL
LIN {X 0,Y 375.983,Z 424.648,A -85,B 0,C 180,E1 -12385.333,E2 -12385.333} C_VEL
LIN {X 0,Y 375.961,Z 424.653,A -85,B 0,C 180,E1 -12388.438,E2 -12388.438} C_VEL
LIN {X 0,Y 375.986,Z 424.652,A -85,B 0,C 180,E1 -12392.14,E2 -12392.14} C_VEL
LIN {X 0,Y 376.008,Z 424.646,A -85,B 0,C 180,E1 -12394.539,E2 -12394.539} C_VEL
LIN {X 0,Y 375.96,Z 424.656,A -85,B 0,C 180,E1 -12398.045,E2 -12398.045} C_VEL
LIN {X 0,Y 376.027,Z 424.645,A -85,B 0,C 180,E1 -12401.474,E2 -12401.474} C_VEL
LIN {X 0,Y 376.063,Z 424.638,A -85,B 0,C 180,E1 -12404.833,E2 -12404.833} C_VEL
LIN {X 0,Y 376.061,Z 424.641,A -85,B 0,C 180,E1 -12408.137,E2 -12408.137} C_VEL
LIN {X 0,Y 376.204,Z 424.625,A -85,B 0,C 180,E1 -12411.938,E2 -12411.938} C_VEL
LIN {X 0,Y 376.173,Z 424.624,A -85,B 0,C 180,E1 -12414.64,E2 -12414.64} C_VEL
LIN {X 0,Y 376.358,Z 424.605,A -85,B 0,C 180,E1 -12417.86,E2 -12417.86} C_VEL
LIN {X 0,Y 376.493,Z 424.587,A -85,B 0,C 180,E1 -12420,E2 -12420} C_VEL
LIN {X 0,Y 376.189,Z 424.625,A -85,B 0,C 180,E1 -12423.213,E2 -12423.213} C_VEL
LIN {X 0,Y 376.218,Z 424.618,A -85,B 0,C 180,E1 -12426.608,E2 -12426.608} C_VEL
LIN {X 0,Y 376.119,Z 424.636,A -85,B 0,C 180,E1 -12429.682,E2 -12429.682} C_VEL
LIN {X 0,Y 376.093,Z 424.638,A -85,B 0,C 180,E1 -12433.658,E2 -12433.658} C_VEL
LIN {X 0,Y 376.047,Z 424.644,A -85,B 0,C 180,E1 -12437.607,E2 -12437.607} C_VEL
LIN {X 0,Y 375.981,Z 424.65,A -85,B 0,C 180,E1 -12440.832,E2 -12440.832} C_VEL
LIN {X 0,Y 375.997,Z 424.646,A -85,B 0,C 180,E1 -12444.281,E2 -12444.281} C_VEL
LIN {X 0,Y 376.023,Z 424.644,A -85,B 0,C 180,E1 -12446.652,E2 -12446.652} C_VEL
LIN {X 0,Y 375.968,Z 424.65,A -85,B 0,C 180,E1 -12450.313,E2 -12450.313} C_VEL
LIN {X 0,Y 375.963,Z 424.65,A -85,B 0,C 180,E1 -12454.111,E2 -12454.111} C_VEL
LIN {X 0,Y 375.956,Z 424.654,A -85,B 0,C 180,E1 -12456.741,E2 -12456.741} C_VEL
LIN {X 0,Y 375.991,Z 424.647,A -85,B 0,C 180,E1 -12459.971,E2 -12459.971} C_VEL
LIN {X 0,Y 375.941,Z 424.654,A -85,B 0,C 180,E1 -12463.765,E2 -12463.765} C_VEL
LIN {X 0,Y 375.992,Z 424.651,A -85,B 0,C 180,E1 -12466.802,E2 -12466.802} C_VEL
LIN {X 0,Y 376.003,Z 424.645,A -85,B 0,C 180,E1 -12470.027,E2 -12470.027} C_VEL
LIN {X 0,Y 375.968,Z 424.651,A -85,B 0,C 180,E1 -12473.495,E2 -12473.495} C_VEL
LIN {X 0,Y 375.963,Z 424.65,A -85,B 0,C 180,E1 -12475.889,E2 -12475.889} C_VEL
LIN {X 0,Y 375.968,Z 424.65,A -85,B 0,C 180,E1 -12479.687,E2 -12479.687} C_VEL
LIN {X 0,Y 376.023,Z 424.645,A -85,B 0,C 180,E1 -12483.348,E2 -12483.348} C_VEL
LIN {X 0,Y 376,Z 424.651,A -85,B 0,C 180,E1 -12486.888,E2 -12486.888} C_VEL
LIN {X 0,Y 376.001,Z 424.648,A -85,B 0,C 180,E1 -12490.339,E2 -12490.339} C_VEL
LIN {X 0,Y 376.062,Z 424.724,A -85,B 0,C 180,E1 -12491.609,E2 -12491.609} C_VEL
LIN {X 0,Y 379.932,Z 436.743,A -85,B 0,C 180,E1 -12492.606,E2 -12492.606} C_VEL
LIN {X 0,Y 382.044,Z 444.277,A -85,B 0,C 180,E1 -12493.345,E2 -12493.345} C_VEL
LIN {X 0,Y 381.251,Z 454.951,A -85,B 0,C 180,E1 -12494.359,E2 -12494.359} C_VEL
LIN {X 0,Y 380.41,Z 465.056,A -85,B 0,C 180,E1 -12495.557,E2 -12495.557} C_VEL
LIN {X 0,Y 379.619,Z 474.099,A -85,B 0,C 180,E1 -12496.892,E2 -12496.892} C_VEL
LIN {X 0,Y 378.602,Z 482.884,A -85,B 0,C 180,E1 -12498.489,E2 -12498.489} C_VEL
LIN {X 0,Y 377.855,Z 489.929,A -85,B 0,C 180,E1 -12500.093,E2 -12500.093} C_VEL
LIN {X 0,Y 377.38,Z 494.668,A -85,B 0,C 180,E1 -12501.432,E2 -12501.432} C_VEL
LIN {X 0,Y 376.882,Z 499.272,A -85,B 0,C 180,E1 -12503.038,E2 -12503.038} C_VEL
LIN {X 0,Y 376.414,Z 502.805,A -85,B 0,C 180,E1 -12504.643,E2 -12504.643} C_VEL
LIN {X 0,Y 376.19,Z 504.627,A -85,B 0,C 180,E1 -12505.714,E2 -12505.714} C_VEL
LIN {X 0,Y 375.994,Z 506.003,A -85,B 0,C 180,E1 -12506.785,E2 -12506.785} C_VEL
LIN {X 0,Y 376.011,Z 507.547,A -85,B 0,C 180,E1 -12508.929,E2 -12508.929} C_VEL
LIN {X 0,Y 376.028,Z 507.77,A -85,B 0,C 180,E1 -12510,E2 -12510} C_VEL
LIN {X 0,Y 376.011,Z 507.59,A -85,B 0,C 180,E1 -12511.071,E2 -12511.071} C_VEL
LIN {X 0,Y 375.988,Z 506.101,A -85,B 0,C 180,E1 -12513.215,E2 -12513.215} C_VEL
LIN {X 0,Y 376.18,Z 504.771,A -85,B 0,C 180,E1 -12514.286,E2 -12514.286} C_VEL
LIN {X 0,Y 376.571,Z 501.957,A -85,B 0,C 180,E1 -12515.892,E2 -12515.892} C_VEL
LIN {X 0,Y 377.094,Z 498.139,A -85,B 0,C 180,E1 -12517.496,E2 -12517.496} C_VEL
LIN {X 0,Y 377.549,Z 492.227,A -85,B 0,C 180,E1 -12519.394,E2 -12519.394} C_VEL
LIN {X 0,Y 378.338,Z 485.841,A -85,B 0,C 180,E1 -12520.976,E2 -12520.976} C_VEL
LIN {X 0,Y 379.26,Z 477.809,A -85,B 0,C 180,E1 -12522.576,E2 -12522.576} C_VEL
LIN {X 0,Y 379.977,Z 469.594,A -85,B 0,C 180,E1 -12523.913,E2 -12523.913} C_VEL
LIN {X 0,Y 380.875,Z 459.406,A -85,B 0,C 180,E1 -12525.245,E2 -12525.245} C_VEL
LIN {X 0,Y 381.748,Z 449.072,A -85,B 0,C 180,E1 -12526.326,E2 -12526.326} C_VEL
LIN {X 0,Y 381.839,Z 443.432,A -85,B 0,C 180,E1 -12526.843,E2 -12526.843} C_VEL
LIN {X 0,Y 378.897,Z 433.527,A -85,B 0,C 180,E1 -12527.786,E2 -12527.786} C_VEL
LIN {X 0,Y 376.026,Z 424.647,A -85,B 0,C 180,E1 -12528.526,E2 -12528.526} C_VEL
LIN {X 0,Y 375.966,Z 424.651,A -85,B 0,C 180,E1 -12531.954,E2 -12531.954} C_VEL
LIN {X 0,Y 376.009,Z 424.649,A -85,B 0,C 180,E1 -12535.461,E2 -12535.461} C_VEL
LIN {X 0,Y 375.963,Z 424.655,A -85,B 0,C 180,E1 -12539.08,E2 -12539.08} C_VEL
LIN {X 0,Y 375.965,Z 424.65,A -85,B 0,C 180,E1 -12540.371,E2 -12540.371} C_VEL
LIN {X 0,Y 375.291,Z 424.74,A -85,B 0,C 180,E1 -12541.265,E2 -12541.265} C_VEL
LIN {X 0,Y 372.468,Z 425.097,A -85,B 0,C 180,E1 -12542.72,E2 -12542.72} C_VEL
LIN {X 0,Y 370.072,Z 425.396,A -85,B 0,C 180,E1 -12543.896,E2 -12543.896} C_VEL
LIN {X 0,Y 369.022,Z 425.522,A -85,B 0,C 180,E1 -12544.805,E2 -12544.805} C_VEL
LIN {X 0,Y 368.924,Z 425.531,A -85,B 0,C 180,E1 -12545.113,E2 -12545.113} C_VEL
LIN {X 0,Y 368.912,Z 425.534,A -85,B 0,C 180,E1 -12548.952,E2 -12548.952} C_VEL
LIN {X 0,Y 368.944,Z 425.524,A -85,B 0,C 180,E1 -12552.02,E2 -12552.02} C_VEL
LIN {X 0,Y 368.927,Z 425.531,A -85,B 0,C 180,E1 -12555.183,E2 -12555.183} C_VEL
LIN {X 0,Y 368.885,Z 425.532,A -85,B 0,C 180,E1 -12558.178,E2 -12558.178} C_VEL
LIN {X 0,Y 368.911,Z 425.531,A -85,B 0,C 180,E1 -12561.36,E2 -12561.36} C_VEL
LIN {X 0,Y 368.938,Z 425.529,A -85,B 0,C 180,E1 -12565.146,E2 -12565.146} C_VEL
LIN {X 0,Y 368.931,Z 425.53,A -85,B 0,C 180,E1 -12569.046,E2 -12569.046} C_VEL
LIN {X 0,Y 368.965,Z 425.528,A -85,B 0,C 180,E1 -12572.797,E2 -12572.797} C_VEL
LIN {X 0,Y 368.947,Z 425.525,A -85,B 0,C 180,E1 -12576.113,E2 -12576.113} C_VEL
LIN {X 0,Y 368.939,Z 425.526,A -85,B 0,C 180,E1 -12579.947,E2 -12579.947} C_VEL
LIN {X 0,Y 368.978,Z 425.52,A -85,B 0,C 180,E1 -12583.399,E2 -12583.399} C_VEL
LIN {X 0,Y 369.062,Z 425.514,A -85,B 0,C 180,E1 -12586.79,E2 -12586.79} C_VEL
LIN {X 0,Y 369.068,Z 425.511,A -85,B 0,C 180,E1 -12590.132,E2 -12590.132} C_VEL
LIN {X 0,Y 369.193,Z 425.493,A -85,B 0,C 180,E1 -12593.441,E2 -12593.441} C_VEL
LIN {X 0,Y 369.322,Z 425.478,A -85,B 0,C 180,E1 -12597.819,E2 -12597.819} C_VEL
LIN {X 0,Y 369.461,Z 425.462,A -85,B 0,C 180,E1 -12600,E2 -12600} C_VEL
LIN {X 0,Y 369.322,Z 425.482,A -85,B 0,C 180,E1 -12602.181,E2 -12602.181} C_VEL
LIN {X 0,Y 369.193,Z 425.497,A -85,B 0,C 180,E1 -12606.558,E2 -12606.558} C_VEL
LIN {X 0,Y 369.068,Z 425.511,A -85,B 0,C 180,E1 -12609.868,E2 -12609.868} C_VEL
LIN {X 0,Y 369.04,Z 425.514,A -85,B 0,C 180,E1 -12613.773,E2 -12613.773} C_VEL
LIN {X 0,Y 369.003,Z 425.519,A -85,B 0,C 180,E1 -12617.768,E2 -12617.768} C_VEL
LIN {X 0,Y 368.911,Z 425.529,A -85,B 0,C 180,E1 -12621.221,E2 -12621.221} C_VEL
LIN {X 0,Y 368.956,Z 425.524,A -85,B 0,C 180,E1 -12624.776,E2 -12624.776} C_VEL
LIN {X 0,Y 368.97,Z 425.521,A -85,B 0,C 180,E1 -12627.203,E2 -12627.203} C_VEL
LIN {X 0,Y 368.931,Z 425.526,A -85,B 0,C 180,E1 -12630.953,E2 -12630.953} C_VEL
LIN {X 0,Y 368.931,Z 425.526,A -85,B 0,C 180,E1 -12635.002,E2 -12635.002} C_VEL
LIN {X 0,Y 368.911,Z 425.529,A -85,B 0,C 180,E1 -12638.641,E2 -12638.641} C_VEL
LIN {X 0,Y 368.883,Z 425.539,A -85,B 0,C 180,E1 -12642.01,E2 -12642.01} C_VEL
LIN {X 0,Y 368.939,Z 425.595,A -85,B 0,C 180,E1 -12644.952,E2 -12644.952} C_VEL
LIN {X 0,Y 370.736,Z 434.462,A -85,B 0,C 180,E1 -12648.433,E2 -12648.433} C_VEL
LIN {X 0,Y 372.34,Z 442.729,A -85,B 0,C 180,E1 -12651.473,E2 -12651.473} C_VEL
LIN {X 0,Y 372.673,Z 446.804,A -85,B 0,C 180,E1 -12652.881,E2 -12652.881} C_VEL
LIN {X 0,Y 371.452,Z 458.739,A -85,B 0,C 180,E1 -12656.723,E2 -12656.723} C_VEL
LIN {X 0,Y 370.729,Z 466.643,A -85,B 0,C 180,E1 -12659.213,E2 -12659.213} C_VEL
LIN {X 0,Y 369.84,Z 478.41,A -85,B 0,C 180,E1 -12662.866,E2 -12662.866} C_VEL
LIN {X 0,Y 369.098,Z 489.972,A -85,B 0,C 180,E1 -12666.43,E2 -12666.43} C_VEL
LIN {X 0,Y 368.48,Z 502.275,A -85,B 0,C 180,E1 -12670.248,E2 -12670.248} C_VEL
LIN {X 0,Y 370.409,Z 518.067,A -85,B 0,C 180,E1 -12670.877,E2 -12670.877} C_VEL
LIN {X 0,Y 371.489,Z 531.572,A -85,B 0,C 180,E1 -12671.633,E2 -12671.633} C_VEL
LIN {X 0,Y 371.851,Z 544.14,A -85,B 0,C 180,E1 -12672.54,E2 -12672.54} C_VEL
LIN {X 0,Y 371.943,Z 552.163,A -85,B 0,C 180,E1 -12673.253,E2 -12673.253} C_VEL
LIN {X 0,Y 370.829,Z 562.645,A -85,B 0,C 180,E1 -12674.332,E2 -12674.332} C_VEL
LIN {X 0,Y 369.852,Z 573.298,A -85,B 0,C 180,E1 -12675.698,E2 -12675.698} C_VEL
LIN {X 0,Y 369.142,Z 581.964,A -85,B 0,C 180,E1 -12677.073,E2 -12677.073} C_VEL
LIN {X 0,Y 368.462,Z 590.439,A -85,B 0,C 180,E1 -12678.726,E2 -12678.726} C_VEL
LIN {X 0,Y 368.124,Z 597.317,A -85,B 0,C 180,E1 -12680.384,E2 -12680.384} C_VEL
LIN {X 0,Y 367.996,Z 603.651,A -85,B 0,C 180,E1 -12682.317,E2 -12682.317} C_VEL
LIN {X 0,Y 368.09,Z 607.794,A -85,B 0,C 180,E1 -12683.972,E2 -12683.972} C_VEL
LIN {X 0,Y 368.293,Z 610.876,A -85,B 0,C 180,E1 -12685.622,E2 -12685.622} C_VEL
LIN {X 0,Y 368.343,Z 612.338,A -85,B 0,C 180,E1 -12686.719,E2 -12686.719} C_VEL
LIN {X 0,Y 368.394,Z 613.382,A -85,B 0,C 180,E1 -12687.813,E2 -12687.813} C_VEL
LIN {X 0,Y 368.709,Z 614.283,A -85,B 0,C 180,E1 -12690,E2 -12690} C_VEL
LIN {X 0,Y 368.394,Z 613.378,A -85,B 0,C 180,E1 -12692.187,E2 -12692.187} C_VEL
LIN {X 0,Y 368.344,Z 612.333,A -85,B 0,C 180,E1 -12693.282,E2 -12693.282} C_VEL
LIN {X 0,Y 368.292,Z 610.868,A -85,B 0,C 180,E1 -12694.378,E2 -12694.378} C_VEL
LIN {X 0,Y 368.086,Z 607.779,A -85,B 0,C 180,E1 -12696.028,E2 -12696.028} C_VEL
LIN {X 0,Y 367.997,Z 603.627,A -85,B 0,C 180,E1 -12697.683,E2 -12697.683} C_VEL
LIN {X 0,Y 368.125,Z 597.286,A -85,B 0,C 180,E1 -12699.616,E2 -12699.616} C_VEL
LIN {X 0,Y 368.462,Z 590.4,A -85,B 0,C 180,E1 -12701.274,E2 -12701.274} C_VEL
LIN {X 0,Y 369.141,Z 581.915,A -85,B 0,C 180,E1 -12702.927,E2 -12702.927} C_VEL
LIN {X 0,Y 369.816,Z 573.229,A -85,B 0,C 180,E1 -12704.303,E2 -12704.303} C_VEL
LIN {X 0,Y 370.772,Z 563.763,A -85,B 0,C 180,E1 -12705.53,E2 -12705.53} C_VEL
LIN {X 0,Y 371.741,Z 553.498,A -85,B 0,C 180,E1 -12706.616,E2 -12706.616} C_VEL
LIN {X 0,Y 372.017,Z 549.023,A -85,B 0,C 180,E1 -12707.027,E2 -12707.027} C_VEL
LIN {X 0,Y 371.687,Z 536.599,A -85,B 0,C 180,E1 -12708.021,E2 -12708.021} C_VEL
LIN {X 0,Y 371.02,Z 524.376,A -85,B 0,C 180,E1 -12708.785,E2 -12708.785} C_VEL
LIN {X 0,Y 369.68,Z 511.388,A -85,B 0,C 180,E1 -12709.401,E2 -12709.401} C_VEL
LIN {X 0,Y 368.483,Z 502.339,A -85,B 0,C 180,E1 -12709.716,E2 -12709.716} C_VEL
LIN {X 0,Y 369.168,Z 488.657,A -85,B 0,C 180,E1 -12713.964,E2 -12713.964} C_VEL
LIN {X 0,Y 369.803,Z 478.364,A -85,B 0,C 180,E1 -12717.137,E2 -12717.137} C_VEL
LIN {X 0,Y 370.868,Z 465.437,A -85,B 0,C 180,E1 -12721.148,E2 -12721.148} C_VEL
LIN {X 0,Y 371.822,Z 454.714,A -85,B 0,C 180,E1 -12724.545,E2 -12724.545} C_VEL
LIN {X 0,Y 372.657,Z 446.755,A -85,B 0,C 180,E1 -12727.121,E2 -12727.121} C_VEL
LIN {X 0,Y 372.314,Z 442.661,A -85,B 0,C 180,E1 -12728.53,E2 -12728.53} C_VEL
LIN {X 0,Y 370.727,Z 434.401,A -85,B 0,C 180,E1 -12731.568,E2 -12731.568} C_VEL
LIN {X 0,Y 368.902,Z 425.532,A -85,B 0,C 180,E1 -12735.069,E2 -12735.069} C_VEL
LIN {X 0,Y 368.886,Z 425.538,A -85,B 0,C 180,E1 -12738.178,E2 -12738.178} C_VEL
LIN {X 0,Y 368.912,Z 425.529,A -85,B 0,C 180,E1 -12741.36,E2 -12741.36} C_VEL
LIN {X 0,Y 368.94,Z 425.525,A -85,B 0,C 180,E1 -12745.147,E2 -12745.147} C_VEL
LIN {X 0,Y 368.932,Z 425.526,A -85,B 0,C 180,E1 -12749.047,E2 -12749.047} C_VEL
LIN {X 0,Y 368.966,Z 425.522,A -85,B 0,C 180,E1 -12752.797,E2 -12752.797} C_VEL
LIN {X 0,Y 368.937,Z 425.53,A -85,B 0,C 180,E1 -12756.117,E2 -12756.117} C_VEL
LIN {X 0,Y 368.94,Z 425.531,A -85,B 0,C 180,E1 -12759.947,E2 -12759.947} C_VEL
LIN {X 0,Y 368.98,Z 425.522,A -85,B 0,C 180,E1 -12763.399,E2 -12763.399} C_VEL
LIN {X 0,Y 369.063,Z 425.51,A -85,B 0,C 180,E1 -12766.79,E2 -12766.79} C_VEL
LIN {X 0,Y 369.069,Z 425.512,A -85,B 0,C 180,E1 -12770.132,E2 -12770.132} C_VEL
LIN {X 0,Y 369.194,Z 425.497,A -85,B 0,C 180,E1 -12773.442,E2 -12773.442} C_VEL
LIN {X 0,Y 369.323,Z 425.482,A -85,B 0,C 180,E1 -12777.819,E2 -12777.819} C_VEL
LIN {X 0,Y 369.462,Z 425.462,A -85,B 0,C 180,E1 -12780,E2 -12780} C_VEL
LIN {X 0,Y 369.321,Z 425.479,A -85,B 0,C 180,E1 -12782.181,E2 -12782.181} C_VEL
LIN {X 0,Y 369.19,Z 425.494,A -85,B 0,C 180,E1 -12786.591,E2 -12786.591} C_VEL
LIN {X 0,Y 369.07,Z 425.512,A -85,B 0,C 180,E1 -12789.868,E2 -12789.868} C_VEL
LIN {X 0,Y 369.041,Z 425.515,A -85,B 0,C 180,E1 -12793.773,E2 -12793.773} C_VEL
LIN {X 0,Y 369.004,Z 425.52,A -85,B 0,C 180,E1 -12797.768,E2 -12797.768} C_VEL
LIN {X 0,Y 368.933,Z 425.531,A -85,B 0,C 180,E1 -12801.22,E2 -12801.22} C_VEL
LIN {X 0,Y 368.961,Z 425.524,A -85,B 0,C 180,E1 -12804.775,E2 -12804.775} C_VEL
LIN {X 0,Y 368.966,Z 425.527,A -85,B 0,C 180,E1 -12807.203,E2 -12807.203} C_VEL
LIN {X 0,Y 368.932,Z 425.529,A -85,B 0,C 180,E1 -12810.953,E2 -12810.953} C_VEL
LIN {X 0,Y 368.932,Z 425.53,A -85,B 0,C 180,E1 -12815.001,E2 -12815.001} C_VEL
LIN {X 0,Y 368.91,Z 425.53,A -85,B 0,C 180,E1 -12818.64,E2 -12818.64} C_VEL
LIN {X 0,Y 368.884,Z 425.532,A -85,B 0,C 180,E1 -12822.009,E2 -12822.009} C_VEL
LIN {X 0,Y 368.958,Z 425.528,A -85,B 0,C 180,E1 -12825.187,E2 -12825.187} C_VEL
LIN {X 0,Y 368.944,Z 425.525,A -85,B 0,C 180,E1 -12828.186,E2 -12828.186} C_VEL
LIN {X 0,Y 368.917,Z 425.53,A -85,B 0,C 180,E1 -12831.359,E2 -12831.359} C_VEL
LIN {X 0,Y 368.94,Z 425.529,A -85,B 0,C 180,E1 -12835.147,E2 -12835.147} C_VEL
LIN {X 0,Y 368.932,Z 425.531,A -85,B 0,C 180,E1 -12839.046,E2 -12839.046} C_VEL
LIN {X 0,Y 368.966,Z 425.528,A -85,B 0,C 180,E1 -12842.797,E2 -12842.797} C_VEL
LIN {X 0,Y 368.948,Z 425.525,A -85,B 0,C 180,E1 -12846.113,E2 -12846.113} C_VEL
LIN {X 0,Y 368.939,Z 425.525,A -85,B 0,C 180,E1 -12849.947,E2 -12849.947} C_VEL
LIN {X 0,Y 368.977,Z 425.525,A -85,B 0,C 180,E1 -12851.224,E2 -12851.224} C_VEL
LIN {X 0,Y 372.516,Z 436.296,A -85,B 0,C 180,E1 -12852.134,E2 -12852.134} C_VEL
LIN {X 0,Y 375.247,Z 445.719,A -85,B 0,C 180,E1 -12853.073,E2 -12853.073} C_VEL
LIN {X 0,Y 374.377,Z 457.229,A -85,B 0,C 180,E1 -12854.205,E2 -12854.205} C_VEL
LIN {X 0,Y 373.61,Z 466.064,A -85,B 0,C 180,E1 -12855.289,E2 -12855.289} C_VEL
LIN {X 0,Y 372.778,Z 475.107,A -85,B 0,C 180,E1 -12856.647,E2 -12856.647} C_VEL
LIN {X 0,Y 371.719,Z 483.891,A -85,B 0,C 180,E1 -12858.273,E2 -12858.273} C_VEL
LIN {X 0,Y 370.935,Z 490.936,A -85,B 0,C 180,E1 -12859.906,E2 -12859.906} C_VEL
LIN {X 0,Y 370.432,Z 495.675,A -85,B 0,C 180,E1 -12861.27,E2 -12861.27} C_VEL
LIN {X 0,Y 369.91,Z 500.278,A -85,B 0,C 180,E1 -12862.906,E2 -12862.906} C_VEL
LIN {X 0,Y 369.418,Z 503.811,A -85,B 0,C 180,E1 -12864.542,E2 -12864.542} C_VEL
LIN {X 0,Y 369.182,Z 505.633,A -85,B 0,C 180,E1 -12865.633,E2 -12865.633} C_VEL
LIN {X 0,Y 368.978,Z 507.008,A -85,B 0,C 180,E1 -12866.724,E2 -12866.724} C_VEL
LIN {X 0,Y 368.997,Z 508.55,A -85,B 0,C 180,E1 -12868.909,E2 -12868.909} C_VEL
LIN {X 0,Y 369.009,Z 508.773,A -85,B 0,C 180,E1 -12870,E2 -12870} C_VEL
LIN {X 0,Y 368.997,Z 508.593,A -85,B 0,C 180,E1 -12871.091,E2 -12871.091} C_VEL
LIN {X 0,Y 368.971,Z 507.106,A -85,B 0,C 180,E1 -12873.276,E2 -12873.276} C_VEL
LIN {X 0,Y 369.172,Z 505.775,A -85,B 0,C 180,E1 -12874.367,E2 -12874.367} C_VEL
LIN {X 0,Y 369.584,Z 502.961,A -85,B 0,C 180,E1 -12876.003,E2 -12876.003} C_VEL
LIN {X 0,Y 370.127,Z 499.143,A -85,B 0,C 180,E1 -12877.638,E2 -12877.638} C_VEL
LIN {X 0,Y 370.617,Z 493.228,A -85,B 0,C 180,E1 -12879.572,E2 -12879.572} C_VEL
LIN {X 0,Y 371.441,Z 486.844,A -85,B 0,C 180,E1 -12881.183,E2 -12881.183} C_VEL
LIN {X 0,Y 372.409,Z 478.811,A -85,B 0,C 180,E1 -12882.811,E2 -12882.811} C_VEL
LIN {X 0,Y 373.159,Z 470.596,A -85,B 0,C 180,E1 -12884.172,E2 -12884.172} C_VEL
LIN {X 0,Y 374.099,Z 460.407,A -85,B 0,C 180,E1 -12885.528,E2 -12885.528} C_VEL
LIN {X 0,Y 375.013,Z 450.071,A -85,B 0,C 180,E1 -12886.628,E2 -12886.628} C_VEL
LIN {X 0,Y 375.034,Z 444.945,A -85,B 0,C 180,E1 -12887.113,E2 -12887.113} C_VEL
LIN {X 0,Y 371.93,Z 434.39,A -85,B 0,C 180,E1 -12888.144,E2 -12888.144} C_VEL
LIN {X 0,Y 368.985,Z 425.524,A -85,B 0,C 180,E1 -12888.893,E2 -12888.893} C_VEL
LIN {X 0,Y 368.935,Z 425.526,A -85,B 0,C 180,E1 -12892.395,E2 -12892.395} C_VEL
LIN {X 0,Y 369.003,Z 425.518,A -85,B 0,C 180,E1 -12895.98,E2 -12895.98} C_VEL
LIN {X 0,Y 368.917,Z 425.53,A -85,B 0,C 180,E1 -12899.69,E2 -12899.69} C_VEL
LIN {X 0,Y 368.901,Z 425.535,A -85,B 0,C 180,E1 -12903.043,E2 -12903.043} C_VEL
LIN {X 0,Y 368.924,Z 425.531,A -85,B 0,C 180,E1 -12905.113,E2 -12905.113} C_VEL
LIN {X 0,Y 368.227,Z 425.614,A -85,B 0,C 180,E1 -12906.024,E2 -12906.024} C_VEL
LIN {X 0,Y 365.381,Z 425.971,A -85,B 0,C 180,E1 -12907.506,E2 -12907.506} C_VEL
LIN {X 0,Y 362.99,Z 426.268,A -85,B 0,C 180,E1 -12908.704,E2 -12908.704} C_VEL
LIN {X 0,Y 361.965,Z 426.395,A -85,B 0,C 180,E1 -12909.631,E2 -12909.631} C_VEL
LIN {X 0,Y 361.881,Z 426.404,A -85,B 0,C 180,E1 -12909.944,E2 -12909.944} C_VEL
LIN {X 0,Y 361.884,Z 426.408,A -85,B 0,C 180,E1 -12912.822,E2 -12912.822} C_VEL
LIN {X 0,Y 361.841,Z 426.409,A -85,B 0,C 180,E1 -12915.943,E2 -12915.943} C_VEL
LIN {X 0,Y 361.838,Z 426.413,A -85,B 0,C 180,E1 -12919.244,E2 -12919.244} C_VEL
LIN {X 0,Y 361.866,Z 426.411,A -85,B 0,C 180,E1 -12922.777,E2 -12922.777} C_VEL
LIN {X 0,Y 361.856,Z 426.407,A -85,B 0,C 180,E1 -12925.72,E2 -12925.72} C_VEL
LIN {X 0,Y 361.875,Z 426.405,A -85,B 0,C 180,E1 -12929.672,E2 -12929.672} C_VEL
LIN {X 0,Y 361.956,Z 426.395,A -85,B 0,C 180,E1 -12933.475,E2 -12933.475} C_VEL
LIN {X 0,Y 361.892,Z 426.405,A -85,B 0,C 180,E1 -12937.145,E2 -12937.145} C_VEL
LIN {X 0,Y 361.909,Z 426.406,A -85,B 0,C 180,E1 -12940.723,E2 -12940.723} C_VEL
LIN {X 0,Y 361.935,Z 426.399,A -85,B 0,C 180,E1 -12943.066,E2 -12943.066} C_VEL
LIN {X 0,Y 362.003,Z 426.395,A -85,B 0,C 180,E1 -12946.528,E2 -12946.528} C_VEL
LIN {X 0,Y 362.034,Z 426.386,A -85,B 0,C 180,E1 -12949.938,E2 -12949.938} C_VEL
LIN {X 0,Y 362.154,Z 426.37,A -85,B 0,C 180,E1 -12953.313,E2 -12953.313} C_VEL
LIN {X 0,Y 362.286,Z 426.354,A -85,B 0,C 180,E1 -12957.776,E2 -12957.776} C_VEL
LIN {X 0,Y 362.431,Z 426.338,A -85,B 0,C 180,E1 -12960,E2 -12960} C_VEL
LIN {X 0,Y 362.286,Z 426.358,A -85,B 0,C 180,E1 -12962.223,E2 -12962.223} C_VEL
LIN {X 0,Y 362.154,Z 426.373,A -85,B 0,C 180,E1 -12966.686,E2 -12966.686} C_VEL
LIN {X 0,Y 362.033,Z 426.389,A -85,B 0,C 180,E1 -12970.062,E2 -12970.062} C_VEL
LIN {X 0,Y 362,Z 426.392,A -85,B 0,C 180,E1 -12973.899,E2 -12973.899} C_VEL
LIN {X 0,Y 361.969,Z 426.397,A -85,B 0,C 180,E1 -12977.939,E2 -12977.939} C_VEL
LIN {X 0,Y 361.863,Z 426.408,A -85,B 0,C 180,E1 -12981.655,E2 -12981.655} C_VEL
LIN {X 0,Y 361.928,Z 426.398,A -85,B 0,C 180,E1 -12985.29,E2 -12985.29} C_VEL
LIN {X 0,Y 361.914,Z 426.404,A -85,B 0,C 180,E1 -12987.779,E2 -12987.779} C_VEL
LIN {X 0,Y 361.84,Z 426.412,A -85,B 0,C 180,E1 -12991.629,E2 -12991.629} C_VEL
LIN {X 0,Y 361.876,Z 426.406,A -85,B 0,C 180,E1 -12995.345,E2 -12995.345} C_VEL
LIN {X 0,Y 361.872,Z 426.405,A -85,B 0,C 180,E1 -12999.027,E2 -12999.027} C_VEL
LIN {X 0,Y 361.838,Z 426.418,A -85,B 0,C 180,E1 -13002.829,E2 -13002.829} C_VEL
LIN {X 0,Y 361.869,Z 426.551,A -85,B 0,C 180,E1 -13004.556,E2 -13004.556} C_VEL
LIN {X 0,Y 363.667,Z 435.275,A -85,B 0,C 180,E1 -13008.075,E2 -13008.075} C_VEL
LIN {X 0,Y 365.169,Z 442.812,A -85,B 0,C 180,E1 -13010.928,E2 -13010.928} C_VEL
LIN {X 0,Y 365.745,Z 446.916,A -85,B 0,C 180,E1 -13012.404,E2 -13012.404} C_VEL
LIN {X 0,Y 364.828,Z 455.847,A -85,B 0,C 180,E1 -13015.37,E2 -13015.37} C_VEL
LIN {X 0,Y 363.93,Z 465.726,A -85,B 0,C 180,E1 -13018.573,E2 -13018.573} C_VEL
LIN {X 0,Y 362.821,Z 478.774,A -85,B 0,C 180,E1 -13022.724,E2 -13022.724} C_VEL
LIN {X 0,Y 361.993,Z 490.868,A -85,B 0,C 180,E1 -13026.547,E2 -13026.547} C_VEL
LIN {X 0,Y 361.437,Z 501.464,A -85,B 0,C 180,E1 -13029.877,E2 -13029.877} C_VEL
LIN {X 0,Y 363.285,Z 515.645,A -85,B 0,C 180,E1 -13030.432,E2 -13030.432} C_VEL
LIN {X 0,Y 364.353,Z 528.161,A -85,B 0,C 180,E1 -13031.112,E2 -13031.112} C_VEL
LIN {X 0,Y 364.83,Z 540.102,A -85,B 0,C 180,E1 -13031.953,E2 -13031.953} C_VEL
LIN {X 0,Y 365.081,Z 551.142,A -85,B 0,C 180,E1 -13032.928,E2 -13032.928} C_VEL
LIN {X 0,Y 363.825,Z 562.817,A -85,B 0,C 180,E1 -13034.166,E2 -13034.166} C_VEL
LIN {X 0,Y 362.906,Z 572.275,A -85,B 0,C 180,E1 -13035.419,E2 -13035.419} C_VEL
LIN {X 0,Y 362.197,Z 580.946,A -85,B 0,C 180,E1 -13036.821,E2 -13036.821} C_VEL
LIN {X 0,Y 361.458,Z 589.419,A -85,B 0,C 180,E1 -13038.504,E2 -13038.504} C_VEL
LIN {X 0,Y 361.071,Z 596.295,A -85,B 0,C 180,E1 -13040.194,E2 -13040.194} C_VEL
LIN {X 0,Y 360.921,Z 602.63,A -85,B 0,C 180,E1 -13042.166,E2 -13042.166} C_VEL
LIN {X 0,Y 361.027,Z 606.779,A -85,B 0,C 180,E1 -13043.854,E2 -13043.854} C_VEL
LIN {X 0,Y 361.223,Z 609.862,A -85,B 0,C 180,E1 -13045.537,E2 -13045.537} C_VEL
LIN {X 0,Y 361.294,Z 611.328,A -85,B 0,C 180,E1 -13046.655,E2 -13046.655} C_VEL
LIN {X 0,Y 361.352,Z 612.375,A -85,B 0,C 180,E1 -13047.771,E2 -13047.771} C_VEL
LIN {X 0,Y 361.681,Z 613.278,A -85,B 0,C 180,E1 -13050,E2 -13050} C_VEL
LIN {X 0,Y 361.353,Z 612.37,A -85,B 0,C 180,E1 -13052.229,E2 -13052.229} C_VEL
LIN {X 0,Y 361.294,Z 611.323,A -85,B 0,C 180,E1 -13053.346,E2 -13053.346} C_VEL
LIN {X 0,Y 361.222,Z 609.853,A -85,B 0,C 180,E1 -13054.464,E2 -13054.464} C_VEL
LIN {X 0,Y 361.025,Z 606.763,A -85,B 0,C 180,E1 -13056.146,E2 -13056.146} C_VEL
LIN {X 0,Y 360.922,Z 602.605,A -85,B 0,C 180,E1 -13057.834,E2 -13057.834} C_VEL
LIN {X 0,Y 361.073,Z 596.261,A -85,B 0,C 180,E1 -13059.806,E2 -13059.806} C_VEL
LIN {X 0,Y 361.458,Z 589.377,A -85,B 0,C 180,E1 -13061.496,E2 -13061.496} C_VEL
LIN {X 0,Y 362.199,Z 580.893,A -85,B 0,C 180,E1 -13063.179,E2 -13063.179} C_VEL
LIN {X 0,Y 362.895,Z 572.204,A -85,B 0,C 180,E1 -13064.582,E2 -13064.582} C_VEL
LIN {X 0,Y 363.823,Z 562.727,A -85,B 0,C 180,E1 -13065.834,E2 -13065.834} C_VEL
LIN {X 0,Y 365.071,Z 551.034,A -85,B 0,C 180,E1 -13067.072,E2 -13067.072} C_VEL
LIN {X 0,Y 364.808,Z 538.745,A -85,B 0,C 180,E1 -13068.144,E2 -13068.144} C_VEL
LIN {X 0,Y 364.217,Z 526.036,A -85,B 0,C 180,E1 -13069.001,E2 -13069.001} C_VEL
LIN {X 0,Y 362.913,Z 512.21,A -85,B 0,C 180,E1 -13069.711,E2 -13069.711} C_VEL
LIN {X 0,Y 361.437,Z 501.216,A -85,B 0,C 180,E1 -13070.144,E2 -13070.144} C_VEL
LIN {X 0,Y 362.146,Z 488.469,A -85,B 0,C 180,E1 -13074.201,E2 -13074.201} C_VEL
LIN {X 0,Y 362.866,Z 477.391,A -85,B 0,C 180,E1 -13077.7,E2 -13077.7} C_VEL
LIN {X 0,Y 364.033,Z 464.372,A -85,B 0,C 180,E1 -13081.847,E2 -13081.847} C_VEL
LIN {X 0,Y 365.175,Z 452.557,A -85,B 0,C 180,E1 -13085.695,E2 -13085.695} C_VEL
LIN {X 0,Y 365.72,Z 446.855,A -85,B 0,C 180,E1 -13087.6,E2 -13087.6} C_VEL
LIN {X 0,Y 364.563,Z 439.639,A -85,B 0,C 180,E1 -13090.232,E2 -13090.232} C_VEL
LIN {X 0,Y 362.879,Z 431.426,A -85,B 0,C 180,E1 -13093.425,E2 -13093.425} C_VEL
LIN {X 0,Y 361.831,Z 426.413,A -85,B 0,C 180,E1 -13095.536,E2 -13095.536} C_VEL
LIN {X 0,Y 361.839,Z 426.417,A -85,B 0,C 180,E1 -13099.244,E2 -13099.244} C_VEL
LIN {X 0,Y 361.868,Z 426.406,A -85,B 0,C 180,E1 -13102.777,E2 -13102.777} C_VEL
LIN {X 0,Y 361.858,Z 426.41,A -85,B 0,C 180,E1 -13105.72,E2 -13105.72} C_VEL
LIN {X 0,Y 361.875,Z 426.408,A -85,B 0,C 180,E1 -13109.672,E2 -13109.672} C_VEL
LIN {X 0,Y 361.957,Z 426.396,A -85,B 0,C 180,E1 -13113.475,E2 -13113.475} C_VEL
LIN {X 0,Y 361.882,Z 426.404,A -85,B 0,C 180,E1 -13117.144,E2 -13117.144} C_VEL
LIN {X 0,Y 361.924,Z 426.399,A -85,B 0,C 180,E1 -13120.724,E2 -13120.724} C_VEL
LIN {X 0,Y 361.95,Z 426.398,A -85,B 0,C 180,E1 -13124.226,E2 -13124.226} C_VEL
LIN {X 0,Y 362.003,Z 426.389,A -85,B 0,C 180,E1 -13126.528,E2 -13126.528} C_VEL
LIN {X 0,Y 362.034,Z 426.389,A -85,B 0,C 180,E1 -13129.938,E2 -13129.938} C_VEL
LIN {X 0,Y 362.155,Z 426.372,A -85,B 0,C 180,E1 -13133.314,E2 -13133.314} C_VEL
LIN {X 0,Y 362.287,Z 426.359,A -85,B 0,C 180,E1 -13137.777,E2 -13137.777} C_VEL
LIN {X 0,Y 362.432,Z 426.338,A -85,B 0,C 180,E1 -13140,E2 -13140} C_VEL
LIN {X 0,Y 362.285,Z 426.355,A -85,B 0,C 180,E1 -13142.224,E2 -13142.224} C_VEL
LIN {X 0,Y 362.154,Z 426.37,A -85,B 0,C 180,E1 -13146.687,E2 -13146.687} C_VEL
LIN {X 0,Y 362.035,Z 426.386,A -85,B 0,C 180,E1 -13150.062,E2 -13150.062} C_VEL
LIN {X 0,Y 362.002,Z 426.391,A -85,B 0,C 180,E1 -13153.899,E2 -13153.899} C_VEL
LIN {X 0,Y 361.97,Z 426.394,A -85,B 0,C 180,E1 -13157.939,E2 -13157.939} C_VEL
LIN {X 0,Y 361.897,Z 426.405,A -85,B 0,C 180,E1 -13161.653,E2 -13161.653} C_VEL
LIN {X 0,Y 361.932,Z 426.404,A -85,B 0,C 180,E1 -13165.29,E2 -13165.29} C_VEL
LIN {X 0,Y 361.911,Z 426.402,A -85,B 0,C 180,E1 -13167.779,E2 -13167.779} C_VEL
LIN {X 0,Y 361.841,Z 426.411,A -85,B 0,C 180,E1 -13171.629,E2 -13171.629} C_VEL
LIN {X 0,Y 361.877,Z 426.409,A -85,B 0,C 180,E1 -13175.345,E2 -13175.345} C_VEL
LIN {X 0,Y 361.872,Z 426.41,A -85,B 0,C 180,E1 -13179.027,E2 -13179.027} C_VEL
LIN {X 0,Y 361.842,Z 426.413,A -85,B 0,C 180,E1 -13182.828,E2 -13182.828} C_VEL
LIN {X 0,Y 361.915,Z 426.4,A -85,B 0,C 180,E1 -13185.931,E2 -13185.931} C_VEL
LIN {X 0,Y 361.908,Z 426.405,A -85,B 0,C 180,E1 -13189.232,E2 -13189.232} C_VEL
LIN {X 0,Y 361.877,Z 426.411,A -85,B 0,C 180,E1 -13192.983,E2 -13192.983} C_VEL
LIN {X 0,Y 361.861,Z 426.41,A -85,B 0,C 180,E1 -13196.631,E2 -13196.631} C_VEL
LIN {X 0,Y 361.876,Z 426.405,A -85,B 0,C 180,E1 -13199.672,E2 -13199.672} C_VEL
LIN {X 0,Y 361.957,Z 426.395,A -85,B 0,C 180,E1 -13203.475,E2 -13203.475} C_VEL
LIN {X 0,Y 361.893,Z 426.405,A -85,B 0,C 180,E1 -13207.145,E2 -13207.145} C_VEL
LIN {X 0,Y 361.939,Z 426.403,A -85,B 0,C 180,E1 -13210.832,E2 -13210.832} C_VEL
LIN {X 0,Y 365.937,Z 438.506,A -85,B 0,C 180,E1 -13211.892,E2 -13211.892} C_VEL
LIN {X 0,Y 368.489,Z 447.45,A -85,B 0,C 180,E1 -13212.819,E2 -13212.819} C_VEL
LIN {X 0,Y 367.621,Z 458.239,A -85,B 0,C 180,E1 -13213.906,E2 -13213.906} C_VEL
LIN {X 0,Y 366.819,Z 467.073,A -85,B 0,C 180,E1 -13215.01,E2 -13215.01} C_VEL
LIN {X 0,Y 365.952,Z 476.113,A -85,B 0,C 180,E1 -13216.393,E2 -13216.393} C_VEL
LIN {X 0,Y 364.842,Z 484.898,A -85,B 0,C 180,E1 -13218.049,E2 -13218.049} C_VEL
LIN {X 0,Y 364.018,Z 491.943,A -85,B 0,C 180,E1 -13219.712,E2 -13219.712} C_VEL
LIN {X 0,Y 363.487,Z 496.682,A -85,B 0,C 180,E1 -13221.102,E2 -13221.102} C_VEL
LIN {X 0,Y 362.94,Z 501.284,A -85,B 0,C 180,E1 -13222.769,E2 -13222.769} C_VEL
LIN {X 0,Y 362.423,Z 504.817,A -85,B 0,C 180,E1 -13224.436,E2 -13224.436} C_VEL
LIN {X 0,Y 362.175,Z 506.639,A -85,B 0,C 180,E1 -13225.548,E2 -13225.548} C_VEL
LIN {X 0,Y 361.962,Z 508.014,A -85,B 0,C 180,E1 -13226.661,E2 -13226.661} C_VEL
LIN {X 0,Y 361.983,Z 509.554,A -85,B 0,C 180,E1 -13228.887,E2 -13228.887} C_VEL
LIN {X 0,Y 361.99,Z 509.777,A -85,B 0,C 180,E1 -13230,E2 -13230} C_VEL
LIN {X 0,Y 361.982,Z 509.596,A -85,B 0,C 180,E1 -13231.112,E2 -13231.112} C_VEL
LIN {X 0,Y 361.955,Z 508.111,A -85,B 0,C 180,E1 -13233.339,E2 -13233.339} C_VEL
LIN {X 0,Y 362.164,Z 506.78,A -85,B 0,C 180,E1 -13234.452,E2 -13234.452} C_VEL
LIN {X 0,Y 362.598,Z 503.965,A -85,B 0,C 180,E1 -13236.119,E2 -13236.119} C_VEL
LIN {X 0,Y 363.162,Z 500.147,A -85,B 0,C 180,E1 -13237.785,E2 -13237.785} C_VEL
LIN {X 0,Y 363.688,Z 494.235,A -85,B 0,C 180,E1 -13239.755,E2 -13239.755} C_VEL
LIN {X 0,Y 364.549,Z 487.847,A -85,B 0,C 180,E1 -13241.397,E2 -13241.397} C_VEL
LIN {X 0,Y 365.562,Z 479.813,A -85,B 0,C 180,E1 -13243.056,E2 -13243.056} C_VEL
LIN {X 0,Y 366.349,Z 471.598,A -85,B 0,C 180,E1 -13244.441,E2 -13244.441} C_VEL
LIN {X 0,Y 367.332,Z 461.408,A -85,B 0,C 180,E1 -13245.821,E2 -13245.821} C_VEL
LIN {X 0,Y 368.311,Z 450.915,A -85,B 0,C 180,E1 -13246.955,E2 -13246.955} C_VEL
LIN {X 0,Y 368.249,Z 446.387,A -85,B 0,C 180,E1 -13247.398,E2 -13247.398} C_VEL
LIN {X 0,Y 364.942,Z 435.395,A -85,B 0,C 180,E1 -13248.507,E2 -13248.507} C_VEL
LIN {X 0,Y 361.923,Z 426.405,A -85,B 0,C 180,E1 -13249.276,E2 -13249.276} C_VEL
LIN {X 0,Y 361.893,Z 426.405,A -85,B 0,C 180,E1 -13252.855,E2 -13252.855} C_VEL
LIN {X 0,Y 361.944,Z 426.398,A -85,B 0,C 180,E1 -13256.721,E2 -13256.721} C_VEL
LIN {X 0,Y 361.875,Z 426.405,A -85,B 0,C 180,E1 -13260.328,E2 -13260.328} C_VEL
LIN {X 0,Y 361.857,Z 426.407,A -85,B 0,C 180,E1 -13264.28,E2 -13264.28} C_VEL
LIN {X 0,Y 361.875,Z 426.41,A -85,B 0,C 180,E1 -13267.225,E2 -13267.225} C_VEL
LIN {X 0,Y 361.881,Z 426.404,A -85,B 0,C 180,E1 -13269.944,E2 -13269.944} C_VEL
LIN {X 0,Y 361.221,Z 426.491,A -85,B 0,C 180,E1 -13270.873,E2 -13270.873} C_VEL
LIN {X 0,Y 358.398,Z 426.839,A -85,B 0,C 180,E1 -13272.385,E2 -13272.385} C_VEL
LIN {X 0,Y 355.991,Z 427.139,A -85,B 0,C 180,E1 -13273.607,E2 -13273.607} C_VEL
LIN {X 0,Y 354.935,Z 427.271,A -85,B 0,C 180,E1 -13274.552,E2 -13274.552} C_VEL
LIN {X 0,Y 354.836,Z 427.282,A -85,B 0,C 180,E1 -13274.872,E2 -13274.872} C_VEL
LIN {X 0,Y 354.79,Z 427.292,A -85,B 0,C 180,E1 -13278.828,E2 -13278.828} C_VEL
LIN {X 0,Y 354.809,Z 427.287,A -85,B 0,C 180,E1 -13282.402,E2 -13282.402} C_VEL
LIN {X 0,Y 354.814,Z 427.29,A -85,B 0,C 180,E1 -13284.941,E2 -13284.941} C_VEL
LIN {X 0,Y 354.795,Z 427.289,A -85,B 0,C 180,E1 -13288.405,E2 -13288.405} C_VEL
LIN {X 0,Y 354.848,Z 427.28,A -85,B 0,C 180,E1 -13291.619,E2 -13291.619} C_VEL
LIN {X 0,Y 354.901,Z 427.275,A -85,B 0,C 180,E1 -13294.173,E2 -13294.173} C_VEL
LIN {X 0,Y 354.837,Z 427.282,A -85,B 0,C 180,E1 -13297.894,E2 -13297.894} C_VEL
LIN {X 0,Y 354.924,Z 427.271,A -85,B 0,C 180,E1 -13301.892,E2 -13301.892} C_VEL
LIN {X 0,Y 354.946,Z 427.269,A -85,B 0,C 180,E1 -13305.981,E2 -13305.981} C_VEL
LIN {X 0,Y 354.982,Z 427.264,A -85,B 0,C 180,E1 -13309.736,E2 -13309.736} C_VEL
LIN {X 0,Y 355.117,Z 427.247,A -85,B 0,C 180,E1 -13313.18,E2 -13313.18} C_VEL
LIN {X 0,Y 355.249,Z 427.231,A -85,B 0,C 180,E1 -13317.732,E2 -13317.732} C_VEL
LIN {X 0,Y 355.4,Z 427.214,A -85,B 0,C 180,E1 -13320,E2 -13320} C_VEL
LIN {X 0,Y 355.249,Z 427.235,A -85,B 0,C 180,E1 -13322.268,E2 -13322.268} C_VEL
LIN {X 0,Y 355.117,Z 427.248,A -85,B 0,C 180,E1 -13326.82,E2 -13326.82} C_VEL
LIN {X 0,Y 354.981,Z 427.27,A -85,B 0,C 180,E1 -13330.264,E2 -13330.264} C_VEL
LIN {X 0,Y 354.946,Z 427.272,A -85,B 0,C 180,E1 -13334.019,E2 -13334.019} C_VEL
LIN {X 0,Y 354.925,Z 427.276,A -85,B 0,C 180,E1 -13338.109,E2 -13338.109} C_VEL
LIN {X 0,Y 354.817,Z 427.29,A -85,B 0,C 180,E1 -13342.107,E2 -13342.107} C_VEL
LIN {X 0,Y 354.9,Z 427.277,A -85,B 0,C 180,E1 -13345.827,E2 -13345.827} C_VEL
LIN {X 0,Y 354.819,Z 427.287,A -85,B 0,C 180,E1 -13349.682,E2 -13349.682} C_VEL
LIN {X 0,Y 354.807,Z 427.289,A -85,B 0,C 180,E1 -13353.702,E2 -13353.702} C_VEL
LIN {X 0,Y 354.801,Z 427.288,A -85,B 0,C 180,E1 -13356.459,E2 -13356.459} C_VEL
LIN {X 0,Y 354.825,Z 427.285,A -85,B 0,C 180,E1 -13359.424,E2 -13359.424} C_VEL
LIN {X 0,Y 354.79,Z 427.296,A -85,B 0,C 180,E1 -13362.867,E2 -13362.867} C_VEL
LIN {X 0,Y 354.808,Z 427.31,A -85,B 0,C 180,E1 -13364.063,E2 -13364.063} C_VEL
LIN {X 0,Y 356.492,Z 435.331,A -85,B 0,C 180,E1 -13367.409,E2 -13367.409} C_VEL
LIN {X 0,Y 358.071,Z 443.444,A -85,B 0,C 180,E1 -13370.567,E2 -13370.567} C_VEL
LIN {X 0,Y 358.737,Z 447.662,A -85,B 0,C 180,E1 -13372.129,E2 -13372.129} C_VEL
LIN {X 0,Y 358.285,Z 452.965,A -85,B 0,C 180,E1 -13373.951,E2 -13373.951} C_VEL
LIN {X 0,Y 357.099,Z 464.8,A -85,B 0,C 180,E1 -13377.901,E2 -13377.901} C_VEL
LIN {X 0,Y 355.824,Z 478.246,A -85,B 0,C 180,E1 -13382.291,E2 -13382.291} C_VEL
LIN {X 0,Y 354.999,Z 490.034,A -85,B 0,C 180,E1 -13386.114,E2 -13386.114} C_VEL
LIN {X 0,Y 354.417,Z 500.258,A -85,B 0,C 180,E1 -13389.449,E2 -13389.449} C_VEL
LIN {X 0,Y 356.356,Z 515.066,A -85,B 0,C 180,E1 -13390.054,E2 -13390.054} C_VEL
LIN {X 0,Y 357.449,Z 528.301,A -85,B 0,C 180,E1 -13390.808,E2 -13390.808} C_VEL
LIN {X 0,Y 357.897,Z 540.248,A -85,B 0,C 180,E1 -13391.688,E2 -13391.688} C_VEL
LIN {X 0,Y 358.108,Z 551.566,A -85,B 0,C 180,E1 -13392.732,E2 -13392.732} C_VEL
LIN {X 0,Y 356.824,Z 562.952,A -85,B 0,C 180,E1 -13393.994,E2 -13393.994} C_VEL
LIN {X 0,Y 355.871,Z 572.361,A -85,B 0,C 180,E1 -13395.299,E2 -13395.299} C_VEL
LIN {X 0,Y 355.251,Z 579.927,A -85,B 0,C 180,E1 -13396.559,E2 -13396.559} C_VEL
LIN {X 0,Y 354.535,Z 587.127,A -85,B 0,C 180,E1 -13397.987,E2 -13397.987} C_VEL
LIN {X 0,Y 354.029,Z 594.222,A -85,B 0,C 180,E1 -13399.708,E2 -13399.708} C_VEL
LIN {X 0,Y 353.887,Z 599.956,A -85,B 0,C 180,E1 -13401.434,E2 -13401.434} C_VEL
LIN {X 0,Y 353.923,Z 605.309,A -85,B 0,C 180,E1 -13403.522,E2 -13403.522} C_VEL
LIN {X 0,Y 354.156,Z 608.849,A -85,B 0,C 180,E1 -13405.447,E2 -13405.447} C_VEL
LIN {X 0,Y 354.245,Z 610.319,A -85,B 0,C 180,E1 -13406.588,E2 -13406.588} C_VEL
LIN {X 0,Y 354.309,Z 611.367,A -85,B 0,C 180,E1 -13407.726,E2 -13407.726} C_VEL
LIN {X 0,Y 354.654,Z 612.273,A -85,B 0,C 180,E1 -13410,E2 -13410} C_VEL
LIN {X 0,Y 354.31,Z 611.362,A -85,B 0,C 180,E1 -13412.274,E2 -13412.274} C_VEL
LIN {X 0,Y 354.245,Z 610.312,A -85,B 0,C 180,E1 -13413.412,E2 -13413.412} C_VEL
LIN {X 0,Y 354.155,Z 608.839,A -85,B 0,C 180,E1 -13414.553,E2 -13414.553} C_VEL
LIN {X 0,Y 353.945,Z 605.293,A -85,B 0,C 180,E1 -13416.476,E2 -13416.476} C_VEL
LIN {X 0,Y 353.888,Z 599.926,A -85,B 0,C 180,E1 -13418.566,E2 -13418.566} C_VEL
LIN {X 0,Y 354.033,Z 594.186,A -85,B 0,C 180,E1 -13420.292,E2 -13420.292} C_VEL
LIN {X 0,Y 354.532,Z 587.08,A -85,B 0,C 180,E1 -13422.014,E2 -13422.014} C_VEL
LIN {X 0,Y 355.248,Z 579.87,A -85,B 0,C 180,E1 -13423.442,E2 -13423.442} C_VEL
LIN {X 0,Y 355.812,Z 572.552,A -85,B 0,C 180,E1 -13424.661,E2 -13424.661} C_VEL
LIN {X 0,Y 356.821,Z 562.863,A -85,B 0,C 180,E1 -13426.007,E2 -13426.007} C_VEL
LIN {X 0,Y 358.107,Z 551.451,A -85,B 0,C 180,E1 -13427.268,E2 -13427.268} C_VEL
LIN {X 0,Y 357.893,Z 539.042,A -85,B 0,C 180,E1 -13428.399,E2 -13428.399} C_VEL
LIN {X 0,Y 357.386,Z 526.757,A -85,B 0,C 180,E1 -13429.279,E2 -13429.279} C_VEL
LIN {X 0,Y 356.166,Z 513.309,A -85,B 0,C 180,E1 -13430.013,E2 -13430.013} C_VEL
LIN {X 0,Y 354.378,Z 500.268,A -85,B 0,C 180,E1 -13430.535,E2 -13430.535} C_VEL
LIN {X 0,Y 355.131,Z 487.926,A -85,B 0,C 180,E1 -13434.557,E2 -13434.557} C_VEL
LIN {X 0,Y 355.963,Z 476.418,A -85,B 0,C 180,E1 -13438.285,E2 -13438.285} C_VEL
LIN {X 0,Y 357.115,Z 464.44,A -85,B 0,C 180,E1 -13442.195,E2 -13442.195} C_VEL
LIN {X 0,Y 358.473,Z 451.557,A -85,B 0,C 180,E1 -13446.503,E2 -13446.503} C_VEL
LIN {X 0,Y 358.705,Z 447.603,A -85,B 0,C 180,E1 -13447.874,E2 -13447.874} C_VEL
LIN {X 0,Y 357.578,Z 440.743,A -85,B 0,C 180,E1 -13450.436,E2 -13450.436} C_VEL
LIN {X 0,Y 355.674,Z 431.396,A -85,B 0,C 180,E1 -13454.176,E2 -13454.176} C_VEL
LIN {X 0,Y 354.8,Z 427.289,A -85,B 0,C 180,E1 -13455.937,E2 -13455.937} C_VEL
LIN {X 0,Y 354.791,Z 427.296,A -85,B 0,C 180,E1 -13459.179,E2 -13459.179} C_VEL
LIN {X 0,Y 354.811,Z 427.288,A -85,B 0,C 180,E1 -13462.402,E2 -13462.402} C_VEL
LIN {X 0,Y 354.815,Z 427.284,A -85,B 0,C 180,E1 -13464.941,E2 -13464.941} C_VEL
LIN {X 0,Y 354.796,Z 427.289,A -85,B 0,C 180,E1 -13468.405,E2 -13468.405} C_VEL
LIN {X 0,Y 354.849,Z 427.283,A -85,B 0,C 180,E1 -13471.619,E2 -13471.619} C_VEL
LIN {X 0,Y 354.901,Z 427.277,A -85,B 0,C 180,E1 -13474.173,E2 -13474.173} C_VEL
LIN {X 0,Y 354.818,Z 427.29,A -85,B 0,C 180,E1 -13477.893,E2 -13477.893} C_VEL
LIN {X 0,Y 354.926,Z 427.276,A -85,B 0,C 180,E1 -13481.891,E2 -13481.891} C_VEL
LIN {X 0,Y 354.947,Z 427.272,A -85,B 0,C 180,E1 -13485.981,E2 -13485.981} C_VEL
LIN {X 0,Y 354.982,Z 427.27,A -85,B 0,C 180,E1 -13489.736,E2 -13489.736} C_VEL
LIN {X 0,Y 355.118,Z 427.248,A -85,B 0,C 180,E1 -13493.18,E2 -13493.18} C_VEL
LIN {X 0,Y 355.25,Z 427.236,A -85,B 0,C 180,E1 -13497.732,E2 -13497.732} C_VEL
LIN {X 0,Y 355.402,Z 427.214,A -85,B 0,C 180,E1 -13500,E2 -13500} C_VEL
LIN {X 0,Y 355.248,Z 427.231,A -85,B 0,C 180,E1 -13502.268,E2 -13502.268} C_VEL
LIN {X 0,Y 355.117,Z 427.247,A -85,B 0,C 180,E1 -13506.82,E2 -13506.82} C_VEL
LIN {X 0,Y 354.983,Z 427.264,A -85,B 0,C 180,E1 -13510.264,E2 -13510.264} C_VEL
LIN {X 0,Y 354.947,Z 427.268,A -85,B 0,C 180,E1 -13514.019,E2 -13514.019} C_VEL
LIN {X 0,Y 354.925,Z 427.27,A -85,B 0,C 180,E1 -13518.108,E2 -13518.108} C_VEL
LIN {X 0,Y 354.839,Z 427.281,A -85,B 0,C 180,E1 -13522.106,E2 -13522.106} C_VEL
LIN {X 0,Y 354.902,Z 427.274,A -85,B 0,C 180,E1 -13525.827,E2 -13525.827} C_VEL
LIN {X 0,Y 354.82,Z 427.285,A -85,B 0,C 180,E1 -13529.682,E2 -13529.682} C_VEL
LIN {X 0,Y 354.809,Z 427.287,A -85,B 0,C 180,E1 -13533.702,E2 -13533.702} C_VEL
LIN {X 0,Y 354.8,Z 427.286,A -85,B 0,C 180,E1 -13536.459,E2 -13536.459} C_VEL
LIN {X 0,Y 354.827,Z 427.286,A -85,B 0,C 180,E1 -13539.424,E2 -13539.424} C_VEL
LIN {X 0,Y 354.794,Z 427.291,A -85,B 0,C 180,E1 -13542.868,E2 -13542.868} C_VEL
LIN {X 0,Y 354.854,Z 427.279,A -85,B 0,C 180,E1 -13546.117,E2 -13546.117} C_VEL
LIN {X 0,Y 354.859,Z 427.283,A -85,B 0,C 180,E1 -13549.189,E2 -13549.189} C_VEL
LIN {X 0,Y 354.816,Z 427.285,A -85,B 0,C 180,E1 -13552.401,E2 -13552.401} C_VEL
LIN {X 0,Y 354.815,Z 427.29,A -85,B 0,C 180,E1 -13554.941,E2 -13554.941} C_VEL
LIN {X 0,Y 354.796,Z 427.288,A -85,B 0,C 180,E1 -13558.405,E2 -13558.405} C_VEL
LIN {X 0,Y 354.849,Z 427.28,A -85,B 0,C 180,E1 -13561.619,E2 -13561.619} C_VEL
LIN {X 0,Y 354.902,Z 427.274,A -85,B 0,C 180,E1 -13564.173,E2 -13564.173} C_VEL
LIN {X 0,Y 354.838,Z 427.282,A -85,B 0,C 180,E1 -13567.894,E2 -13567.894} C_VEL
LIN {X 0,Y 354.87,Z 427.281,A -85,B 0,C 180,E1 -13570.42,E2 -13570.42} C_VEL
LIN {X 0,Y 359.08,Z 439.875,A -85,B 0,C 180,E1 -13571.559,E2 -13571.559} C_VEL
LIN {X 0,Y 361.581,Z 448.514,A -85,B 0,C 180,E1 -13572.482,E2 -13572.482} C_VEL
LIN {X 0,Y 361.543,Z 452.096,A -85,B 0,C 180,E1 -13572.84,E2 -13572.84} C_VEL
LIN {X 0,Y 360.545,Z 462.73,A -85,B 0,C 180,E1 -13574.018,E2 -13574.018} C_VEL
LIN {X 0,Y 359.637,Z 471.926,A -85,B 0,C 180,E1 -13575.283,E2 -13575.283} C_VEL
LIN {X 0,Y 358.752,Z 480.29,A -85,B 0,C 180,E1 -13576.692,E2 -13576.692} C_VEL
LIN {X 0,Y 357.667,Z 488.42,A -85,B 0,C 180,E1 -13578.381,E2 -13578.381} C_VEL
LIN {X 0,Y 356.868,Z 494.544,A -85,B 0,C 180,E1 -13579.959,E2 -13579.959} C_VEL
LIN {X 0,Y 356.398,Z 499.341,A -85,B 0,C 180,E1 -13581.495,E2 -13581.495} C_VEL
LIN {X 0,Y 355.72,Z 503.588,A -85,B 0,C 180,E1 -13583.192,E2 -13583.192} C_VEL
LIN {X 0,Y 355.429,Z 505.823,A -85,B 0,C 180,E1 -13584.326,E2 -13584.326} C_VEL
LIN {X 0,Y 355.168,Z 507.645,A -85,B 0,C 180,E1 -13585.46,E2 -13585.46} C_VEL
LIN {X 0,Y 354.946,Z 509.02,A -85,B 0,C 180,E1 -13586.594,E2 -13586.594} C_VEL
LIN {X 0,Y 354.967,Z 510.558,A -85,B 0,C 180,E1 -13588.865,E2 -13588.865} C_VEL
LIN {X 0,Y 354.97,Z 510.781,A -85,B 0,C 180,E1 -13590,E2 -13590} C_VEL
LIN {X 0,Y 354.966,Z 510.599,A -85,B 0,C 180,E1 -13591.134,E2 -13591.134} C_VEL
LIN {X 0,Y 354.939,Z 509.115,A -85,B 0,C 180,E1 -13593.405,E2 -13593.405} C_VEL
LIN {X 0,Y 355.157,Z 507.784,A -85,B 0,C 180,E1 -13594.54,E2 -13594.54} C_VEL
LIN {X 0,Y 355.613,Z 504.969,A -85,B 0,C 180,E1 -13596.24,E2 -13596.24} C_VEL
LIN {X 0,Y 356.2,Z 501.15,A -85,B 0,C 180,E1 -13597.939,E2 -13597.939} C_VEL
LIN {X 0,Y 356.763,Z 495.242,A -85,B 0,C 180,E1 -13599.945,E2 -13599.945} C_VEL
LIN {X 0,Y 357.663,Z 488.849,A -85,B 0,C 180,E1 -13601.619,E2 -13601.619} C_VEL
LIN {X 0,Y 358.721,Z 480.815,A -85,B 0,C 180,E1 -13603.309,E2 -13603.309} C_VEL
LIN {X 0,Y 359.547,Z 472.599,A -85,B 0,C 180,E1 -13604.721,E2 -13604.721} C_VEL
LIN {X 0,Y 360.576,Z 462.409,A -85,B 0,C 180,E1 -13606.126,E2 -13606.126} C_VEL
LIN {X 0,Y 361.528,Z 452.401,A -85,B 0,C 180,E1 -13607.233,E2 -13607.233} C_VEL
LIN {X 0,Y 361.732,Z 449.511,A -85,B 0,C 180,E1 -13607.518,E2 -13607.518} C_VEL
LIN {X 0,Y 359.063,Z 439.748,A -85,B 0,C 180,E1 -13608.557,E2 -13608.557} C_VEL
LIN {X 0,Y 354.875,Z 427.282,A -85,B 0,C 180,E1 -13609.712,E2 -13609.712} C_VEL
LIN {X 0,Y 354.835,Z 427.288,A -85,B 0,C 180,E1 -13613.336,E2 -13613.336} C_VEL
LIN {X 0,Y 354.89,Z 427.279,A -85,B 0,C 180,E1 -13616.981,E2 -13616.981} C_VEL
LIN {X 0,Y 354.82,Z 427.285,A -85,B 0,C 180,E1 -13619.682,E2 -13619.682} C_VEL
LIN {X 0,Y 354.808,Z 427.286,A -85,B 0,C 180,E1 -13623.702,E2 -13623.702} C_VEL
LIN {X 0,Y 354.804,Z 427.286,A -85,B 0,C 180,E1 -13626.459,E2 -13626.459} C_VEL
LIN {X 0,Y 354.814,Z 427.284,A -85,B 0,C 180,E1 -13629.945,E2 -13629.945} C_VEL
LIN {X 0,Y 354.837,Z 427.286,A -85,B 0,C 180,E1 -13632.875,E2 -13632.875} C_VEL
LIN {X 0,Y 354.836,Z 427.282,A -85,B 0,C 180,E1 -13634.872,E2 -13634.872} C_VEL
LIN {X 0,Y 354.127,Z 427.371,A -85,B 0,C 180,E1 -13635.82,E2 -13635.82} C_VEL
LIN {X 0,Y 351.238,Z 427.732,A -85,B 0,C 180,E1 -13637.361,E2 -13637.361} C_VEL
LIN {X 0,Y 348.826,Z 428.033,A -85,B 0,C 180,E1 -13638.608,E2 -13638.608} C_VEL
LIN {X 0,Y 347.811,Z 428.158,A -85,B 0,C 180,E1 -13639.573,E2 -13639.573} C_VEL
LIN {X 0,Y 347.738,Z 428.166,A -85,B 0,C 180,E1 -13639.9,E2 -13639.9} C_VEL
LIN {X 0,Y 347.764,Z 428.167,A -85,B 0,C 180,E1 -13642.679,E2 -13642.679} C_VEL
LIN {X 0,Y 347.75,Z 428.165,A -85,B 0,C 180,E1 -13645.956,E2 -13645.956} C_VEL
LIN {X 0,Y 347.751,Z 428.164,A -85,B 0,C 180,E1 -13649.652,E2 -13649.652} C_VEL
LIN {X 0,Y 347.833,Z 428.154,A -85,B 0,C 180,E1 -13653.608,E2 -13653.608} C_VEL
LIN {X 0,Y 347.791,Z 428.16,A -85,B 0,C 180,E1 -13656.162,E2 -13656.162} C_VEL
LIN {X 0,Y 347.815,Z 428.157,A -85,B 0,C 180,E1 -13659.909,E2 -13659.909} C_VEL
LIN {X 0,Y 347.868,Z 428.153,A -85,B 0,C 180,E1 -13662.359,E2 -13662.359} C_VEL
LIN {X 0,Y 347.9,Z 428.147,A -85,B 0,C 180,E1 -13665.971,E2 -13665.971} C_VEL
LIN {X 0,Y 347.933,Z 428.141,A -85,B 0,C 180,E1 -13669.526,E2 -13669.526} C_VEL
LIN {X 0,Y 348.085,Z 428.124,A -85,B 0,C 180,E1 -13673.042,E2 -13673.042} C_VEL
LIN {X 0,Y 348.211,Z 428.107,A -85,B 0,C 180,E1 -13677.686,E2 -13677.686} C_VEL
LIN {X 0,Y 348.37,Z 428.089,A -85,B 0,C 180,E1 -13680,E2 -13680} C_VEL
LIN {X 0,Y 348.211,Z 428.112,A -85,B 0,C 180,E1 -13682.313,E2 -13682.313} C_VEL
LIN {X 0,Y 348.082,Z 428.123,A -85,B 0,C 180,E1 -13686.958,E2 -13686.958} C_VEL
LIN {X 0,Y 347.932,Z 428.146,A -85,B 0,C 180,E1 -13690.474,E2 -13690.474} C_VEL
LIN {X 0,Y 347.9,Z 428.151,A -85,B 0,C 180,E1 -13694.15,E2 -13694.15} C_VEL
LIN {X 0,Y 347.893,Z 428.152,A -85,B 0,C 180,E1 -13698.291,E2 -13698.291} C_VEL
LIN {X 0,Y 347.769,Z 428.164,A -85,B 0,C 180,E1 -13701.626,E2 -13701.626} C_VEL
LIN {X 0,Y 347.813,Z 428.157,A -85,B 0,C 180,E1 -13705.108,E2 -13705.108} C_VEL
LIN {X 0,Y 347.811,Z 428.16,A -85,B 0,C 180,E1 -13707.694,E2 -13707.694} C_VEL
LIN {X 0,Y 347.751,Z 428.167,A -85,B 0,C 180,E1 -13710.348,E2 -13710.348} C_VEL
LIN {X 0,Y 347.75,Z 428.17,A -85,B 0,C 180,E1 -13714.044,E2 -13714.044} C_VEL
LIN {X 0,Y 347.764,Z 428.164,A -85,B 0,C 180,E1 -13717.321,E2 -13717.321} C_VEL
LIN {X 0,Y 347.734,Z 428.17,A -85,B 0,C 180,E1 -13720.297,E2 -13720.297} C_VEL
LIN {X 0,Y 347.728,Z 428.177,A -85,B 0,C 180,E1 -13723.607,E2 -13723.607} C_VEL
LIN {X 0,Y 349.587,Z 436.897,A -85,B 0,C 180,E1 -13727.33,E2 -13727.33} C_VEL
LIN {X 0,Y 351.266,Z 445.566,A -85,B 0,C 180,E1 -13730.771,E2 -13730.771} C_VEL
LIN {X 0,Y 351.815,Z 450.092,A -85,B 0,C 180,E1 -13732.463,E2 -13732.463} C_VEL
LIN {X 0,Y 350.419,Z 461.887,A -85,B 0,C 180,E1 -13736.527,E2 -13736.527} C_VEL
LIN {X 0,Y 349.38,Z 471.84,A -85,B 0,C 180,E1 -13739.88,E2 -13739.88} C_VEL
LIN {X 0,Y 348.444,Z 483.166,A -85,B 0,C 180,E1 -13743.658,E2 -13743.658} C_VEL
